# B&R Automation Studio project TD52 (part 70)

```iecst
END_TYPE
TYPE
END_TYPE
```

#### lib_properties.txt
```
For manual assignment to hardware configuration please
add the following additional include directories:

\Logical\MATLAB_includes\R2021b\

And the following additional build options:

-lm -D MODEL=Gen2_ref -D NUMST=1 -D NCSTATES=0 -D HAVESTDIO -D MODEL_HAS_DYNAMICALLY_LOADED_SFCNS=0 -D CLASSIC_INTERFACE=0 -D ALLOCATIONFCN=0 -D TID01EQ=0 -D TERMFCN=1 -D ONESTEPFCN=1 -D MAT_FILE=0 -D MULTI_INSTANCE_CODE=1 -D INTEGER_CODE=0 -D MT=0
```

#### rtGetInf.c
```c
/********************************************************************
 * COPYRIGHT -- B&R Industrial Automation GmbH
 ********************************************************************
 * Program: Gen2_ref
 * File: rtGetInf.c
 * Author: 105055527
 * Last modified by: kelleto00
 * Created: Wed Apr 16 13:02:53 2008
 * Last modified: Wed Oct 09 10:01:33 2024
 * Model Version: 4.14.00.04
 * Description: V4.10.00.01, 01-09-2020 Keller, Ke Estimator, additive LS factor, Ptraj SpeedCtrl, LVRT Freeze HLCi
   V4.10.00.01, 02-10-2020 Keller, bugfix HLCi p2srefLX init, BDC_lib: change Inf to 1e7
   V4.10.00.01, 13-11-2020 Keller, bugfix LXcorr T2s/ZZP, LSLff damping, dbgOut for Leanox WG compensation
   V4.10.00.01, 27-01-2021 Keller, Lx WGV compensation: no reset in island mode, addition before skipfire compensation
   V4.10.00.01, 02-02-2021 Keller, initialization lambda estimation with rLam_Start
   V4.11.00.01, 28-05-2021 Keller, Gas Quality Change (GQC) Improvements, LHV estimator output
   V4.11.00.01, 05-11-2021 Keller, Bugfix BDC: worksplit offset, optionally Nset instead of Nnom, rN_Eng_LRskipF
   V4.12.00.01, 10-02-2021 Keller, SpeedCtrl2.0 TU Wien: Disturbance Estimator, LQR incl. droop & leanox
   V4.12.00.02, 23-05-2022 Arnold, Leanox point C in low load
   V4.12.00.02, 09-06-2022 Kafka, add external skip fire input for isolated and grid parallel operation
   V4.12.00.03, 15-09-2022 Keller, add power trajectory to HLCi for extended LQR (Droop setpoint)
   V4.12.00.04, 12-10-2022 Keller, add gas flow comp. factor for rejections
   V4.12.00.05, 13-10-2022 Keller, power filter for static skipfire in island mode
   V4.12.00.06, 15-11-2022 Keller, Ke adaptation with disturbance observer
   V4.13.00.01, 15-11-2022 Keller, FDC: R_mix output, HLCi: R_mix for Ke
   V4.13.00.02, 10-07-2023 Keller, interpolation of LHV, rho_gas and Lmin
   V4.13.00.03, 10-07-2023 Keller, load dependent gas dosage delay
   V4.13.00.04, 11-09-2023 Keller, D-part FSM, bugfix dPTV ramp
   V4.13.00.05, 27-02-2024 Keller, Filter outputs without bSS
   V4.13.00.06, 10-04-2024 Keller, bugfix leanox manual mode with bSepEmisCtrl
   V4.14.00.01, 01-07-2024 Keller, iNskip_LRfor Ke calculation
   V4.14.00.02, 17-09-2024 Keller, Use actual speed for observer disturbance dg (Gen2_ref/HLC_Island (HLC_Island_ref)/iLQR_SF/Ref LQR)
   V4.14.00.03, 30-09-2024 Keller, LR gas flow compensation possible without actuator saturation
   V4.14.00.04, 02-10-2024 Keller, Limit derivative power setpoint for FSM
 * modified Comment:
 ********************************************************************
 * Implementation of program Gen2_ref
 ********************************************************************
 * Generated with B&R Automation Studio Target for Simulink V6.7.1
 * (ERT based)
 ********************************************************************/

/*
 * Abstract:
 *      Function to initialize non-finite, Inf
 */
#include "rtGetInf.h"

/*  Defines */
#define NumBitsPerChar                 8U

/*  Data Types */

/**************************** GLOBAL DATA *************************************/
/*  Definitions */

/*  Declarations  */

/***************************** FILE SCOPE DATA ********************************/

/*************************** FUNCTIONS ****************************************/

/*
 * Initialize rtInf needed by the generated code.
 * Inf is initialized as non-signaling. Assumes IEEE.
 */
real_T rtGetInf(void)
{
  size_t bitsPerReal = sizeof(real_T) * (NumBitsPerChar);
  real_T inf = 0.0;
  if (bitsPerReal == 32U) {
    inf = rtGetInfF();
  } else {
    union {
      LittleEndianIEEEDouble bitVal;
      real_T fltVal;
    } tmpVal;

    tmpVal.bitVal.words.wordH = 0x7FF00000U;
    tmpVal.bitVal.words.wordL = 0x00000000U;
    inf = tmpVal.fltVal;
  }

  return inf;
}

/*
 * Initialize rtInfF needed by the generated code.
 * Inf is initialized as non-signaling. Assumes IEEE.
 */
real32_T rtGetInfF(void)
{
  IEEESingle infF;
  infF.wordL.wordLuint = 0x7F800000U;
  return infF.wordL.wordLreal;
}

/*
 * Initialize rtMinusInf needed by the generated code.
 * Inf is initialized as non-signaling. Assumes IEEE.
 */
real_T rtGetMinusInf(void)
{
  size_t bitsPerReal = sizeof(real_T) * (NumBitsPerChar);
  real_T minf = 0.0;
  if (bitsPerReal == 32U) {
    minf = rtGetMinusInfF();
  } else {
    union {
      LittleEndianIEEEDouble bitVal;
      real_T fltVal;
    } tmpVal;

    tmpVal.bitVal.words.wordH = 0xFFF00000U;
    tmpVal.bitVal.words.wordL = 0x00000000U;
    minf = tmpVal.fltVal;
  }

  return minf;
}

/*
 * Initialize rtMinusInfF needed by the generated code.
 * Inf is initialized as non-signaling. Assumes IEEE.
 */
real32_T rtGetMinusInfF(void)
{
  IEEESingle minfF;
  minfF.wordL.wordLuint = 0xFF800000U;
  return minfF.wordL.wordLreal;
}

/*======================== TOOL VERSION INFORMATION ==========================*
 * MATLAB 9.11 (R2021b)14-May-2021                                            *
 * Simulink 10.4 (R2021b)14-May-2021                                          *
 * Simulink Coder 9.6 (R2021b)14-May-2021                                     *
 * Embedded Coder 7.7 (R2021b)14-May-2021                                     *
 * Stateflow 10.5 (R2021b)14-May-2021                                         *
 *============================================================================*/

/*======================= LICENSE IN USE INFORMATION =========================*
 * control_toolbox                                                            *
 * matlab                                                                     *
 * matlab_coder                                                               *
 * real-time_workshop                                                         *
 * rtw_embedded_coder                                                         *
 * simulink                                                                   *
 *============================================================================*/
```

#### rtGetInf.h
```c
/********************************************************************
 * COPYRIGHT -- B&R Industrial Automation GmbH
 ********************************************************************
 * Program: Gen2_ref
 * File: rtGetInf.h
 * Author: 105055527
 * Last modified by: kelleto00
 * Created: Wed Apr 16 13:02:53 2008
 * Last modified: Wed Oct 09 10:01:33 2024
 * Model Version: 4.14.00.04
 * Description: V4.10.00.01, 01-09-2020 Keller, Ke Estimator, additive LS factor, Ptraj SpeedCtrl, LVRT Freeze HLCi
   V4.10.00.01, 02-10-2020 Keller, bugfix HLCi p2srefLX init, BDC_lib: change Inf to 1e7
   V4.10.00.01, 13-11-2020 Keller, bugfix LXcorr T2s/ZZP, LSLff damping, dbgOut for Leanox WG compensation
   V4.10.00.01, 27-01-2021 Keller, Lx WGV compensation: no reset in island mode, addition before skipfire compensation
   V4.10.00.01, 02-02-2021 Keller, initialization lambda estimation with rLam_Start
   V4.11.00.01, 28-05-2021 Keller, Gas Quality Change (GQC) Improvements, LHV estimator output
   V4.11.00.01, 05-11-2021 Keller, Bugfix BDC: worksplit offset, optionally Nset instead of Nnom, rN_Eng_LRskipF
   V4.12.00.01, 10-02-2021 Keller, SpeedCtrl2.0 TU Wien: Disturbance Estimator, LQR incl. droop & leanox
   V4.12.00.02, 23-05-2022 Arnold, Leanox point C in low load
   V4.12.00.02, 09-06-2022 Kafka, add external skip fire input for isolated and grid parallel operation
   V4.12.00.03, 15-09-2022 Keller, add power trajectory to HLCi for extended LQR (Droop setpoint)
   V4.12.00.04, 12-10-2022 Keller, add gas flow comp. factor for rejections
   V4.12.00.05, 13-10-2022 Keller, power filter for static skipfire in island mode
   V4.12.00.06, 15-11-2022 Keller, Ke adaptation with disturbance observer
   V4.13.00.01, 15-11-2022 Keller, FDC: R_mix output, HLCi: R_mix for Ke
   V4.13.00.02, 10-07-2023 Keller, interpolation of LHV, rho_gas and Lmin
   V4.13.00.03, 10-07-2023 Keller, load dependent gas dosage delay
   V4.13.00.04, 11-09-2023 Keller, D-part FSM, bugfix dPTV ramp
   V4.13.00.05, 27-02-2024 Keller, Filter outputs without bSS
   V4.13.00.06, 10-04-2024 Keller, bugfix leanox manual mode with bSepEmisCtrl
   V4.14.00.01, 01-07-2024 Keller, iNskip_LRfor Ke calculation
   V4.14.00.02, 17-09-2024 Keller, Use actual speed for observer disturbance dg (Gen2_ref/HLC_Island (HLC_Island_ref)/iLQR_SF/Ref LQR)
   V4.14.00.03, 30-09-2024 Keller, LR gas flow compensation possible without actuator saturation
   V4.14.00.04, 02-10-2024 Keller, Limit derivative power setpoint for FSM
 * modified Comment:
 ********************************************************************
 * Header for program Gen2_ref
 ********************************************************************
 * Generated with B&R Automation Studio Target for Simulink V6.7.1
 * (ERT based)
 ********************************************************************/

#ifndef RTW_HEADER_rtGetInf_h_
#define RTW_HEADER_rtGetInf_h_
#include <stddef.h>
#include "rtwtypes.h"
#include "rt_nonfinite.h"
#ifndef MIN
#define MIN(a,b)                       ((a) < (b) ? (a) : (b))
#endif

#ifndef MAX
#define MAX(a,b)                       ((a) > (b) ? (a) : (b))
#endif

#ifndef AST_ROUND
#define AST_ROUND(x)                   ((x)>=0?(long long)((x)+0.5):(long long)((x)-0.5))
#endif

extern real_T rtGetInf(void);
extern real32_T rtGetInfF(void);
extern real_T rtGetMinusInf(void);
extern real32_T rtGetMinusInfF(void);

#endif                                 /* RTW_HEADER_rtGetInf_h_ */
```

#### rtGetNaN.c
```c
/********************************************************************
 * COPYRIGHT -- B&R Industrial Automation GmbH
 ********************************************************************
 * Program: Gen2_ref
 * File: rtGetNaN.c
 * Author: 105055527
 * Last modified by: kelleto00
 * Created: Wed Apr 16 13:02:53 2008
 * Last modified: Wed Oct 09 10:01:33 2024
 * Model Version: 4.14.00.04
 * Description: V4.10.00.01, 01-09-2020 Keller, Ke Estimator, additive LS factor, Ptraj SpeedCtrl, LVRT Freeze HLCi
   V4.10.00.01, 02-10-2020 Keller, bugfix HLCi p2srefLX init, BDC_lib: change Inf to 1e7
   V4.10.00.01, 13-11-2020 Keller, bugfix LXcorr T2s/ZZP, LSLff damping, dbgOut for Leanox WG compensation
   V4.10.00.01, 27-01-2021 Keller, Lx WGV compensation: no reset in island mode, addition before skipfire compensation
   V4.10.00.01, 02-02-2021 Keller, initialization lambda estimation with rLam_Start
   V4.11.00.01, 28-05-2021 Keller, Gas Quality Change (GQC) Improvements, LHV estimator output
   V4.11.00.01, 05-11-2021 Keller, Bugfix BDC: worksplit offset, optionally Nset instead of Nnom, rN_Eng_LRskipF
   V4.12.00.01, 10-02-2021 Keller, SpeedCtrl2.0 TU Wien: Disturbance Estimator, LQR incl. droop & leanox
   V4.12.00.02, 23-05-2022 Arnold, Leanox point C in low load
   V4.12.00.02, 09-06-2022 Kafka, add external skip fire input for isolated and grid parallel operation
   V4.12.00.03, 15-09-2022 Keller, add power trajectory to HLCi for extended LQR (Droop setpoint)
   V4.12.00.04, 12-10-2022 Keller, add gas flow comp. factor for rejections
   V4.12.00.05, 13-10-2022 Keller, power filter for static skipfire in island mode
   V4.12.00.06, 15-11-2022 Keller, Ke adaptation with disturbance observer
   V4.13.00.01, 15-11-2022 Keller, FDC: R_mix output, HLCi: R_mix for Ke
   V4.13.00.02, 10-07-2023 Keller, interpolation of LHV, rho_gas and Lmin
   V4.13.00.03, 10-07-2023 Keller, load dependent gas dosage delay
   V4.13.00.04, 11-09-2023 Keller, D-part FSM, bugfix dPTV ramp
   V4.13.00.05, 27-02-2024 Keller, Filter outputs without bSS
   V4.13.00.06, 10-04-2024 Keller, bugfix leanox manual mode with bSepEmisCtrl
   V4.14.00.01, 01-07-2024 Keller, iNskip_LRfor Ke calculation
   V4.14.00.02, 17-09-2024 Keller, Use actual speed for observer disturbance dg (Gen2_ref/HLC_Island (HLC_Island_ref)/iLQR_SF/Ref LQR)
   V4.14.00.03, 30-09-2024 Keller, LR gas flow compensation possible without actuator saturation
   V4.14.00.04, 02-10-2024 Keller, Limit derivative power setpoint for FSM
 * modified Comment:
 ********************************************************************
 * Implementation of program Gen2_ref
 ********************************************************************
 * Generated with B&R Automation Studio Target for Simulink V6.7.1
 * (ERT based)
 ********************************************************************/

/*
 * Abstract:
 *      Function to initialize non-finite, NaN
 */
#include "rtGetNaN.h"

/*  Defines */
#define NumBitsPerChar                 8U

/*  Data Types */

/**************************** GLOBAL DATA *************************************/
/*  Definitions */

/*  Declarations  */

/***************************** FILE SCOPE DATA ********************************/

/*************************** FUNCTIONS ****************************************/

/*
 * Initialize rtNaN needed by the generated code.
 * NaN is initialized as non-signaling. Assumes IEEE.
 */
real_T rtGetNaN(void)
{
  size_t bitsPerReal = sizeof(real_T) * (NumBitsPerChar);
  real_T nan = 0.0;
  if (bitsPerReal == 32U) {
    nan = rtGetNaNF();
  } else {
    union {
      LittleEndianIEEEDouble bitVal;
      real_T fltVal;
    } tmpVal;

    tmpVal.bitVal.words.wordH = 0xFFF80000U;
    tmpVal.bitVal.words.wordL = 0x00000000U;
    nan = tmpVal.fltVal;
  }

  return nan;
}

/*
 * Initialize rtNaNF needed by the generated code.
 * NaN is initialized as non-signaling. Assumes IEEE.
 */
real32_T rtGetNaNF(void)
{
  IEEESingle nanF = { { 0.0F } };

  nanF.wordL.wordLuint = 0xFFC00000U;
  return nanF.wordL.wordLreal;
}

/*======================== TOOL VERSION INFORMATION ==========================*
 * MATLAB 9.11 (R2021b)14-May-2021                                            *
 * Simulink 10.4 (R2021b)14-May-2021                                          *
 * Simulink Coder 9.6 (R2021b)14-May-2021                                     *
 * Embedded Coder 7.7 (R2021b)14-May-2021                                     *
 * Stateflow 10.5 (R2021b)14-May-2021                                         *
 *============================================================================*/

/*======================= LICENSE IN USE INFORMATION =========================*
 * control_toolbox                                                            *
 * matlab                                                                     *
 * matlab_coder                                                               *
 * real-time_workshop                                                         *
 * rtw_embedded_coder                                                         *
 * simulink                                                                   *
 *============================================================================*/
```

#### rtGetNaN.h
```c
/********************************************************************
 * COPYRIGHT -- B&R Industrial Automation GmbH
 ********************************************************************
 * Program: Gen2_ref
 * File: rtGetNaN.h
 * Author: 105055527
 * Last modified by: kelleto00
 * Created: Wed Apr 16 13:02:53 2008
 * Last modified: Wed Oct 09 10:01:33 2024
 * Model Version: 4.14.00.04
 * Description: V4.10.00.01, 01-09-2020 Keller, Ke Estimator, additive LS factor, Ptraj SpeedCtrl, LVRT Freeze HLCi
   V4.10.00.01, 02-10-2020 Keller, bugfix HLCi p2srefLX init, BDC_lib: change Inf to 1e7
   V4.10.00.01, 13-11-2020 Keller, bugfix LXcorr T2s/ZZP, LSLff damping, dbgOut for Leanox WG compensation
   V4.10.00.01, 27-01-2021 Keller, Lx WGV compensation: no reset in island mode, addition before skipfire compensation
   V4.10.00.01, 02-02-2021 Keller, initialization lambda estimation with rLam_Start
   V4.11.00.01, 28-05-2021 Keller, Gas Quality Change (GQC) Improvements, LHV estimator output
   V4.11.00.01, 05-11-2021 Keller, Bugfix BDC: worksplit offset, optionally Nset instead of Nnom, rN_Eng_LRskipF
   V4.12.00.01, 10-02-2021 Keller, SpeedCtrl2.0 TU Wien: Disturbance Estimator, LQR incl. droop & leanox
   V4.12.00.02, 23-05-2022 Arnold, Leanox point C in low load
   V4.12.00.02, 09-06-2022 Kafka, add external skip fire input for isolated and grid parallel operation
   V4.12.00.03, 15-09-2022 Keller, add power trajectory to HLCi for extended LQR (Droop setpoint)
   V4.12.00.04, 12-10-2022 Keller, add gas flow comp. factor for rejections
   V4.12.00.05, 13-10-2022 Keller, power filter for static skipfire in island mode
   V4.12.00.06, 15-11-2022 Keller, Ke adaptation with disturbance observer
   V4.13.00.01, 15-11-2022 Keller, FDC: R_mix output, HLCi: R_mix for Ke
   V4.13.00.02, 10-07-2023 Keller, interpolation of LHV, rho_gas and Lmin
   V4.13.00.03, 10-07-2023 Keller, load dependent gas dosage delay
   V4.13.00.04, 11-09-2023 Keller, D-part FSM, bugfix dPTV ramp
   V4.13.00.05, 27-02-2024 Keller, Filter outputs without bSS
   V4.13.00.06, 10-04-2024 Keller, bugfix leanox manual mode with bSepEmisCtrl
   V4.14.00.01, 01-07-2024 Keller, iNskip_LRfor Ke calculation
   V4.14.00.02, 17-09-2024 Keller, Use actual speed for observer disturbance dg (Gen2_ref/HLC_Island (HLC_Island_ref)/iLQR_SF/Ref LQR)
   V4.14.00.03, 30-09-2024 Keller, LR gas flow compensation possible without actuator saturation
   V4.14.00.04, 02-10-2024 Keller, Limit derivative power setpoint for FSM
 * modified Comment:
 ********************************************************************
 * Header for program Gen2_ref
 ********************************************************************
 * Generated with B&R Automation Studio Target for Simulink V6.7.1
 * (ERT based)
 ********************************************************************/

#ifndef RTW_HEADER_rtGetNaN_h_
#define RTW_HEADER_rtGetNaN_h_
#include <stddef.h>
#include "rtwtypes.h"
#include "rt_nonfinite.h"
#ifndef MIN
#define MIN(a,b)                       ((a) < (b) ? (a) : (b))
#endif

#ifndef MAX
#define MAX(a,b)                       ((a) > (b) ? (a) : (b))
#endif

#ifndef AST_ROUND
#define AST_ROUND(x)                   ((x)>=0?(long long)((x)+0.5):(long long)((x)-0.5))
#endif

extern real_T rtGetNaN(void);
extern real32_T rtGetNaNF(void);

#endif                                 /* RTW_HEADER_rtGetNaN_h_ */
```

#### rt_defines.h
```c
/********************************************************************
 * COPYRIGHT -- B&R Industrial Automation GmbH
 ********************************************************************
 * Program: Gen2_ref
 * File: rt_defines.h
 * Author: 105055527
 * Last modified by: kelleto00
 * Created: Wed Apr 16 13:02:53 2008
 * Last modified: Wed Oct 09 10:01:33 2024
 * Model Version: 4.14.00.04
 * Description: V4.10.00.01, 01-09-2020 Keller, Ke Estimator, additive LS factor, Ptraj SpeedCtrl, LVRT Freeze HLCi
   V4.10.00.01, 02-10-2020 Keller, bugfix HLCi p2srefLX init, BDC_lib: change Inf to 1e7
   V4.10.00.01, 13-11-2020 Keller, bugfix LXcorr T2s/ZZP, LSLff damping, dbgOut for Leanox WG compensation
   V4.10.00.01, 27-01-2021 Keller, Lx WGV compensation: no reset in island mode, addition before skipfire compensation
   V4.10.00.01, 02-02-2021 Keller, initialization lambda estimation with rLam_Start
   V4.11.00.01, 28-05-2021 Keller, Gas Quality Change (GQC) Improvements, LHV estimator output
   V4.11.00.01, 05-11-2021 Keller, Bugfix BDC: worksplit offset, optionally Nset instead of Nnom, rN_Eng_LRskipF
   V4.12.00.01, 10-02-2021 Keller, SpeedCtrl2.0 TU Wien: Disturbance Estimator, LQR incl. droop & leanox
   V4.12.00.02, 23-05-2022 Arnold, Leanox point C in low load
   V4.12.00.02, 09-06-2022 Kafka, add external skip fire input for isolated and grid parallel operation
   V4.12.00.03, 15-09-2022 Keller, add power trajectory to HLCi for extended LQR (Droop setpoint)
   V4.12.00.04, 12-10-2022 Keller, add gas flow comp. factor for rejections
   V4.12.00.05, 13-10-2022 Keller, power filter for static skipfire in island mode
   V4.12.00.06, 15-11-2022 Keller, Ke adaptation with disturbance observer
   V4.13.00.01, 15-11-2022 Keller, FDC: R_mix output, HLCi: R_mix for Ke
   V4.13.00.02, 10-07-2023 Keller, interpolation of LHV, rho_gas and Lmin
   V4.13.00.03, 10-07-2023 Keller, load dependent gas dosage delay
   V4.13.00.04, 11-09-2023 Keller, D-part FSM, bugfix dPTV ramp
   V4.13.00.05, 27-02-2024 Keller, Filter outputs without bSS
   V4.13.00.06, 10-04-2024 Keller, bugfix leanox manual mode with bSepEmisCtrl
   V4.14.00.01, 01-07-2024 Keller, iNskip_LRfor Ke calculation
   V4.14.00.02, 17-09-2024 Keller, Use actual speed for observer disturbance dg (Gen2_ref/HLC_Island (HLC_Island_ref)/iLQR_SF/Ref LQR)
   V4.14.00.03, 30-09-2024 Keller, LR gas flow compensation possible without actuator saturation
   V4.14.00.04, 02-10-2024 Keller, Limit derivative power setpoint for FSM
 * modified Comment:
 ********************************************************************
 * Header for program Gen2_ref
 ********************************************************************
 * Generated with B&R Automation Studio Target for Simulink V6.7.1
 * (ERT based)
 ********************************************************************/

#ifndef RTW_HEADER_rt_defines_h_
#define RTW_HEADER_rt_defines_h_
#ifndef MIN
#define MIN(a,b)                       ((a) < (b) ? (a) : (b))
#endif

#ifndef MAX
#define MAX(a,b)                       ((a) > (b) ? (a) : (b))
#endif

#ifndef AST_ROUND
#define AST_ROUND(x)                   ((x)>=0?(long long)((x)+0.5):(long long)((x)-0.5))
#endif

/*===========*
 * Constants *
 *===========*/
#define RT_PI                          3.14159265358979323846
#define RT_PIF                         3.1415927F
#define RT_LN_10                       2.30258509299404568402
#define RT_LN_10F                      2.3025851F
#define RT_LOG10E                      0.43429448190325182765
#define RT_LOG10EF                     0.43429449F
#define RT_E                           2.7182818284590452354
#define RT_EF                          2.7182817F

/*
 * UNUSED_PARAMETER(x)
 *   Used to specify that a function parameter (argument) is required but not
 *   accessed by the function body.
 */
#ifndef UNUSED_PARAMETER
#if defined(__LCC__)
#define UNUSED_PARAMETER(x)                                      /* do nothing */
#else

/*
 * This is the semi-ANSI standard way of indicating that an
 * unused function parameter is required.
 */
#define UNUSED_PARAMETER(x)            (void) (x)
#endif
#endif
#endif                                 /* RTW_HEADER_rt_defines_h_ */
```

#### rt_nonfinite.c
```c
/********************************************************************
 * COPYRIGHT -- B&R Industrial Automation GmbH
 ********************************************************************
 * Program: Gen2_ref
 * File: rt_nonfinite.c
 * Author: 105055527
 * Last modified by: kelleto00
 * Created: Wed Apr 16 13:02:53 2008
 * Last modified: Wed Oct 09 10:01:33 2024
 * Model Version: 4.14.00.04
 * Description: V4.10.00.01, 01-09-2020 Keller, Ke Estimator, additive LS factor, Ptraj SpeedCtrl, LVRT Freeze HLCi
   V4.10.00.01, 02-10-2020 Keller, bugfix HLCi p2srefLX init, BDC_lib: change Inf to 1e7
   V4.10.00.01, 13-11-2020 Keller, bugfix LXcorr T2s/ZZP, LSLff damping, dbgOut for Leanox WG compensation
   V4.10.00.01, 27-01-2021 Keller, Lx WGV compensation: no reset in island mode, addition before skipfire compensation
   V4.10.00.01, 02-02-2021 Keller, initialization lambda estimation with rLam_Start
   V4.11.00.01, 28-05-2021 Keller, Gas Quality Change (GQC) Improvements, LHV estimator output
   V4.11.00.01, 05-11-2021 Keller, Bugfix BDC: worksplit offset, optionally Nset instead of Nnom, rN_Eng_LRskipF
   V4.12.00.01, 10-02-2021 Keller, SpeedCtrl2.0 TU Wien: Disturbance Estimator, LQR incl. droop & leanox
   V4.12.00.02, 23-05-2022 Arnold, Leanox point C in low load
   V4.12.00.02, 09-06-2022 Kafka, add external skip fire input for isolated and grid parallel operation
   V4.12.00.03, 15-09-2022 Keller, add power trajectory to HLCi for extended LQR (Droop setpoint)
   V4.12.00.04, 12-10-2022 Keller, add gas flow comp. factor for rejections
   V4.12.00.05, 13-10-2022 Keller, power filter for static skipfire in island mode
   V4.12.00.06, 15-11-2022 Keller, Ke adaptation with disturbance observer
   V4.13.00.01, 15-11-2022 Keller, FDC: R_mix output, HLCi: R_mix for Ke
   V4.13.00.02, 10-07-2023 Keller, interpolation of LHV, rho_gas and Lmin
   V4.13.00.03, 10-07-2023 Keller, load dependent gas dosage delay
   V4.13.00.04, 11-09-2023 Keller, D-part FSM, bugfix dPTV ramp
   V4.13.00.05, 27-02-2024 Keller, Filter outputs without bSS
   V4.13.00.06, 10-04-2024 Keller, bugfix leanox manual mode with bSepEmisCtrl
   V4.14.00.01, 01-07-2024 Keller, iNskip_LRfor Ke calculation
   V4.14.00.02, 17-09-2024 Keller, Use actual speed for observer disturbance dg (Gen2_ref/HLC_Island (HLC_Island_ref)/iLQR_SF/Ref LQR)
   V4.14.00.03, 30-09-2024 Keller, LR gas flow compensation possible without actuator saturation
   V4.14.00.04, 02-10-2024 Keller, Limit derivative power setpoint for FSM
 * modified Comment:
 ********************************************************************
 * Implementation of program Gen2_ref
 ********************************************************************
 * Generated with B&R Automation Studio Target for Simulink V6.7.1
 * (ERT based)
 ********************************************************************/

/*
 * Abstract:
 *      Function to initialize non-finites,
 *      (Inf, NaN and -Inf).
 */
#include "rt_nonfinite.h"
#include "rtGetNaN.h"
#include "rtGetInf.h"

/*  Defines */
#define NumBitsPerChar                 8U

/*  Data Types */

/**************************** GLOBAL DATA *************************************/
/*  Definitions */

/*  Declarations  */
real_T rtInf;
real_T rtMinusInf;
real_T rtNaN;
real32_T rtInfF;
real32_T rtMinusInfF;
real32_T rtNaNF;

/***************************** FILE SCOPE DATA ********************************/

/*************************** FUNCTIONS ****************************************/

/*
 * Initialize the rtInf, rtMinusInf, and rtNaN needed by the
 * generated code. NaN is initialized as non-signaling. Assumes IEEE.
 */
void rt_InitInfAndNaN(size_t realSize)
{
  (void) (realSize);
  rtNaN = rtGetNaN();
  rtNaNF = rtGetNaNF();
  rtInf = rtGetInf();
  rtInfF = rtGetInfF();
  rtMinusInf = rtGetMinusInf();
  rtMinusInfF = rtGetMinusInfF();
}

/* Test if value is infinite */
boolean_T rtIsInf(real_T value)
{
  return (boolean_T)((value==rtInf || value==rtMinusInf) ? 1U : 0U);
}

/* Test if single-precision value is infinite */
boolean_T rtIsInfF(real32_T value)
{
  return (boolean_T)(((value)==rtInfF || (value)==rtMinusInfF) ? 1U : 0U);
}

/* Test if value is not a number */
boolean_T rtIsNaN(real_T value)
{
  boolean_T result = (boolean_T) 0;
  size_t bitsPerReal = sizeof(real_T) * (NumBitsPerChar);
  if (bitsPerReal == 32U) {
    result = rtIsNaNF((real32_T)value);
  } else {
    union {
      LittleEndianIEEEDouble bitVal;
      real_T fltVal;
    } tmpVal;

    tmpVal.fltVal = value;
    result = (boolean_T)((tmpVal.bitVal.words.wordH & 0x7FF00000) == 0x7FF00000 &&
                         ( (tmpVal.bitVal.words.wordH & 0x000FFFFF) != 0 ||
                          (tmpVal.bitVal.words.wordL != 0) ));
  }

  return result;
}

/* Test if single-precision value is not a number */
boolean_T rtIsNaNF(real32_T value)
{
  IEEESingle tmp;
  tmp.wordL.wordLreal = value;
  return (boolean_T)( (tmp.wordL.wordLuint & 0x7F800000) == 0x7F800000 &&
                     (tmp.wordL.wordLuint & 0x007FFFFF) != 0 );
}

/*======================== TOOL VERSION INFORMATION ==========================*
 * MATLAB 9.11 (R2021b)14-May-2021                                            *
 * Simulink 10.4 (R2021b)14-May-2021                                          *
 * Simulink Coder 9.6 (R2021b)14-May-2021                                     *
 * Embedded Coder 7.7 (R2021b)14-May-2021                                     *
 * Stateflow 10.5 (R2021b)14-May-2021                                         *
 *============================================================================*/

/*======================= LICENSE IN USE INFORMATION =========================*
 * control_toolbox                                                            *
 * matlab                                                                     *
 * matlab_coder                                                               *
 * real-time_workshop                                                         *
 * rtw_embedded_coder                                                         *
 * simulink                                                                   *
 *============================================================================*/
```

#### rt_nonfinite.h
```c
/********************************************************************
 * COPYRIGHT -- B&R Industrial Automation GmbH
 ********************************************************************
 * Program: Gen2_ref
 * File: rt_nonfinite.h
 * Author: 105055527
 * Last modified by: kelleto00
 * Created: Wed Apr 16 13:02:53 2008
 * Last modified: Wed Oct 09 10:01:33 2024
 * Model Version: 4.14.00.04
 * Description: V4.10.00.01, 01-09-2020 Keller, Ke Estimator, additive LS factor, Ptraj SpeedCtrl, LVRT Freeze HLCi
   V4.10.00.01, 02-10-2020 Keller, bugfix HLCi p2srefLX init, BDC_lib: change Inf to 1e7
   V4.10.00.01, 13-11-2020 Keller, bugfix LXcorr T2s/ZZP, LSLff damping, dbgOut for Leanox WG compensation
   V4.10.00.01, 27-01-2021 Keller, Lx WGV compensation: no reset in island mode, addition before skipfire compensation
   V4.10.00.01, 02-02-2021 Keller, initialization lambda estimation with rLam_Start
   V4.11.00.01, 28-05-2021 Keller, Gas Quality Change (GQC) Improvements, LHV estimator output
   V4.11.00.01, 05-11-2021 Keller, Bugfix BDC: worksplit offset, optionally Nset instead of Nnom, rN_Eng_LRskipF
   V4.12.00.01, 10-02-2021 Keller, SpeedCtrl2.0 TU Wien: Disturbance Estimator, LQR incl. droop & leanox
   V4.12.00.02, 23-05-2022 Arnold, Leanox point C in low load
   V4.12.00.02, 09-06-2022 Kafka, add external skip fire input for isolated and grid parallel operation
   V4.12.00.03, 15-09-2022 Keller, add power trajectory to HLCi for extended LQR (Droop setpoint)
   V4.12.00.04, 12-10-2022 Keller, add gas flow comp. factor for rejections
   V4.12.00.05, 13-10-2022 Keller, power filter for static skipfire in island mode
   V4.12.00.06, 15-11-2022 Keller, Ke adaptation with disturbance observer
   V4.13.00.01, 15-11-2022 Keller, FDC: R_mix output, HLCi: R_mix for Ke
   V4.13.00.02, 10-07-2023 Keller, interpolation of LHV, rho_gas and Lmin
   V4.13.00.03, 10-07-2023 Keller, load dependent gas dosage delay
   V4.13.00.04, 11-09-2023 Keller, D-part FSM, bugfix dPTV ramp
   V4.13.00.05, 27-02-2024 Keller, Filter outputs without bSS
   V4.13.00.06, 10-04-2024 Keller, bugfix leanox manual mode with bSepEmisCtrl
   V4.14.00.01, 01-07-2024 Keller, iNskip_LRfor Ke calculation
   V4.14.00.02, 17-09-2024 Keller, Use actual speed for observer disturbance dg (Gen2_ref/HLC_Island (HLC_Island_ref)/iLQR_SF/Ref LQR)
   V4.14.00.03, 30-09-2024 Keller, LR gas flow compensation possible without actuator saturation
   V4.14.00.04, 02-10-2024 Keller, Limit derivative power setpoint for FSM
 * modified Comment:
 ********************************************************************
 * Header for program Gen2_ref
 ********************************************************************
 * Generated with B&R Automation Studio Target for Simulink V6.7.1
 * (ERT based)
 ********************************************************************/

#ifndef RTW_HEADER_rt_nonfinite_h_
#define RTW_HEADER_rt_nonfinite_h_
#include <stddef.h>
#include "rtwtypes.h"
#ifndef MIN
#define MIN(a,b)                       ((a) < (b) ? (a) : (b))
#endif

#ifndef MAX
#define MAX(a,b)                       ((a) > (b) ? (a) : (b))
#endif

#ifndef AST_ROUND
#define AST_ROUND(x)                   ((x)>=0?(long long)((x)+0.5):(long long)((x)-0.5))
#endif

extern real_T rtInf;
extern real_T rtMinusInf;
extern real_T rtNaN;
extern real32_T rtInfF;
extern real32_T rtMinusInfF;
extern real32_T rtNaNF;
extern void rt_InitInfAndNaN(size_t realSize);
extern boolean_T rtIsInf(real_T value);
extern boolean_T rtIsInfF(real32_T value);
extern boolean_T rtIsNaN(real_T value);
extern boolean_T rtIsNaNF(real32_T value);
typedef struct {
  struct {
    uint32_T wordH;
    uint32_T wordL;
  } words;
} BigEndianIEEEDouble;

typedef struct {
  struct {
    uint32_T wordL;
    uint32_T wordH;
  } words;
} LittleEndianIEEEDouble;

typedef struct {
  union {
    real32_T wordLreal;
    uint32_T wordLuint;
  } wordL;
} IEEESingle;

#endif                                 /* RTW_HEADER_rt_nonfinite_h_ */
```

#### rtwtypes.h
```c
/********************************************************************
 * COPYRIGHT -- B&R Industrial Automation GmbH
 ********************************************************************
 * Program: Gen2_ref
 * File: rtwtypes.h
 * Author: 105055527
 * Last modified by: kelleto00
 * Created: Wed Apr 16 13:02:53 2008
 * Last modified: Wed Oct 09 10:01:33 2024
 * Model Version: 4.14.00.04
 * Description: V4.10.00.01, 01-09-2020 Keller, Ke Estimator, additive LS factor, Ptraj SpeedCtrl, LVRT Freeze HLCi
   V4.10.00.01, 02-10-2020 Keller, bugfix HLCi p2srefLX init, BDC_lib: change Inf to 1e7
   V4.10.00.01, 13-11-2020 Keller, bugfix LXcorr T2s/ZZP, LSLff damping, dbgOut for Leanox WG compensation
   V4.10.00.01, 27-01-2021 Keller, Lx WGV compensation: no reset in island mode, addition before skipfire compensation
   V4.10.00.01, 02-02-2021 Keller, initialization lambda estimation with rLam_Start
   V4.11.00.01, 28-05-2021 Keller, Gas Quality Change (GQC) Improvements, LHV estimator output
   V4.11.00.01, 05-11-2021 Keller, Bugfix BDC: worksplit offset, optionally Nset instead of Nnom, rN_Eng_LRskipF
   V4.12.00.01, 10-02-2021 Keller, SpeedCtrl2.0 TU Wien: Disturbance Estimator, LQR incl. droop & leanox
   V4.12.00.02, 23-05-2022 Arnold, Leanox point C in low load
   V4.12.00.02, 09-06-2022 Kafka, add external skip fire input for isolated and grid parallel operation
   V4.12.00.03, 15-09-2022 Keller, add power trajectory to HLCi for extended LQR (Droop setpoint)
   V4.12.00.04, 12-10-2022 Keller, add gas flow comp. factor for rejections
   V4.12.00.05, 13-10-2022 Keller, power filter for static skipfire in island mode
   V4.12.00.06, 15-11-2022 Keller, Ke adaptation with disturbance observer
   V4.13.00.01, 15-11-2022 Keller, FDC: R_mix output, HLCi: R_mix for Ke
   V4.13.00.02, 10-07-2023 Keller, interpolation of LHV, rho_gas and Lmin
   V4.13.00.03, 10-07-2023 Keller, load dependent gas dosage delay
   V4.13.00.04, 11-09-2023 Keller, D-part FSM, bugfix dPTV ramp
   V4.13.00.05, 27-02-2024 Keller, Filter outputs without bSS
   V4.13.00.06, 10-04-2024 Keller, bugfix leanox manual mode with bSepEmisCtrl
   V4.14.00.01, 01-07-2024 Keller, iNskip_LRfor Ke calculation
   V4.14.00.02, 17-09-2024 Keller, Use actual speed for observer disturbance dg (Gen2_ref/HLC_Island (HLC_Island_ref)/iLQR_SF/Ref LQR)
   V4.14.00.03, 30-09-2024 Keller, LR gas flow compensation possible without actuator saturation
   V4.14.00.04, 02-10-2024 Keller, Limit derivative power setpoint for FSM
 * modified Comment:
 ********************************************************************
 * Header for program Gen2_ref
 ********************************************************************
 * Generated with B&R Automation Studio Target for Simulink V6.7.1
 * (ERT based)
 ********************************************************************/

#ifndef RTWTYPES_H
#define RTWTYPES_H

/* Logical type definitions */
#if (!defined(__cplusplus))
#ifndef false
#define false                          (0U)
#endif

#ifndef true
#define true                           (1U)
#endif
#endif

/*=======================================================================*
 * Target hardware information
 *   Device type: Intel->x86/Pentium
 *   Number of bits:     char:   8    short:   16    long:  32
 *                       long:  32
 *                       native word size:  32
 *   Byte ordering: LittleEndian
 *   Signed integer division rounds to: Zero
 *   Shift right on a signed integer as arithmetic shift: on
 *=======================================================================*/

/*=======================================================================*
 * Fixed width word size data types:                                     *
 *   int8_T, int16_T, int32_T     - signed 8, 16, or 32 bit integers     *
 *   uint8_T, uint16_T, uint32_T  - unsigned 8, 16, or 32 bit integers   *
 *   real32_T, real64_T           - 32 and 64 bit floating point numbers *
 *=======================================================================*/
typedef signed char int8_T;
typedef unsigned char uint8_T;
typedef short int16_T;
typedef unsigned short uint16_T;
typedef long int32_T;
typedef unsigned long uint32_T;
typedef float real32_T;
typedef double real64_T;

/*===========================================================================*
 * Generic type definitions: boolean_T, char_T, byte_T, int_T, uint_T,       *
 *                           real_T, time_T, ulong_T.                        *
 *===========================================================================*/
typedef double real_T;
typedef double time_T;
typedef unsigned char boolean_T;
typedef long int_T;
typedef unsigned long uint_T;
typedef unsigned long ulong_T;
typedef char char_T;
typedef unsigned char uchar_T;
typedef char_T byte_T;

/*=======================================================================*
 * Min and Max:                                                          *
 *   int8_T, int16_T, int32_T     - signed 8, 16, or 32 bit integers     *
 *   uint8_T, uint16_T, uint32_T  - unsigned 8, 16, or 32 bit integers   *
 *=======================================================================*/
#define MAX_int8_T                     ((int8_T)(127))
#define MIN_int8_T                     ((int8_T)(-128))
#define MAX_uint8_T                    ((uint8_T)(255U))
#define MAX_int16_T                    ((int16_T)(32767))
#define MIN_int16_T                    ((int16_T)(-32768))
#define MAX_uint16_T                   ((uint16_T)(65535U))
#define MAX_int32_T                    ((int32_T)(2147483647))
#define MIN_int32_T                    ((int32_T)(-2147483647-1))
#define MAX_uint32_T                   ((uint32_T)(0xFFFFFFFFU))

/* Block D-Work pointer type */
typedef void * pointer_T;

#endif                                 /* RTWTYPES_H */

#ifndef MIN
#define MIN(a,b)                       ((a) < (b) ? (a) : (b))
#endif

#ifndef MAX
#define MAX(a,b)                       ((a) > (b) ? (a) : (b))
#endif

#ifndef AST_ROUND
#define AST_ROUND(x)                   ((x)>=0?(long long)((x)+0.5):(long long)((x)-0.5))
#endif
```

#### zero_crossing_types.h
```c
/********************************************************************
 * COPYRIGHT -- B&R Industrial Automation GmbH
 ********************************************************************
 * Program: Gen2_ref
 * File: zero_crossing_types.h
 * Author: 105055527
 * Last modified by: kelleto00
 * Created: Wed Apr 16 13:02:53 2008
 * Last modified: Wed Oct 09 10:01:33 2024
 * Model Version: 4.14.00.04
 * Description: V4.10.00.01, 01-09-2020 Keller, Ke Estimator, additive LS factor, Ptraj SpeedCtrl, LVRT Freeze HLCi
   V4.10.00.01, 02-10-2020 Keller, bugfix HLCi p2srefLX init, BDC_lib: change Inf to 1e7
   V4.10.00.01, 13-11-2020 Keller, bugfix LXcorr T2s/ZZP, LSLff damping, dbgOut for Leanox WG compensation
   V4.10.00.01, 27-01-2021 Keller, Lx WGV compensation: no reset in island mode, addition before skipfire compensation
   V4.10.00.01, 02-02-2021 Keller, initialization lambda estimation with rLam_Start
   V4.11.00.01, 28-05-2021 Keller, Gas Quality Change (GQC) Improvements, LHV estimator output
   V4.11.00.01, 05-11-2021 Keller, Bugfix BDC: worksplit offset, optionally Nset instead of Nnom, rN_Eng_LRskipF
   V4.12.00.01, 10-02-2021 Keller, SpeedCtrl2.0 TU Wien: Disturbance Estimator, LQR incl. droop & leanox
   V4.12.00.02, 23-05-2022 Arnold, Leanox point C in low load
   V4.12.00.02, 09-06-2022 Kafka, add external skip fire input for isolated and grid parallel operation
   V4.12.00.03, 15-09-2022 Keller, add power trajectory to HLCi for extended LQR (Droop setpoint)
   V4.12.00.04, 12-10-2022 Keller, add gas flow comp. factor for rejections
   V4.12.00.05, 13-10-2022 Keller, power filter for static skipfire in island mode
   V4.12.00.06, 15-11-2022 Keller, Ke adaptation with disturbance observer
   V4.13.00.01, 15-11-2022 Keller, FDC: R_mix output, HLCi: R_mix for Ke
   V4.13.00.02, 10-07-2023 Keller, interpolation of LHV, rho_gas and Lmin
   V4.13.00.03, 10-07-2023 Keller, load dependent gas dosage delay
   V4.13.00.04, 11-09-2023 Keller, D-part FSM, bugfix dPTV ramp
   V4.13.00.05, 27-02-2024 Keller, Filter outputs without bSS
   V4.13.00.06, 10-04-2024 Keller, bugfix leanox manual mode with bSepEmisCtrl
   V4.14.00.01, 01-07-2024 Keller, iNskip_LRfor Ke calculation
   V4.14.00.02, 17-09-2024 Keller, Use actual speed for observer disturbance dg (Gen2_ref/HLC_Island (HLC_Island_ref)/iLQR_SF/Ref LQR)
   V4.14.00.03, 30-09-2024 Keller, LR gas flow compensation possible without actuator saturation
   V4.14.00.04, 02-10-2024 Keller, Limit derivative power setpoint for FSM
 * modified Comment:
 ********************************************************************
 * Header for program Gen2_ref
 ********************************************************************
 * Generated with B&R Automation Studio Target for Simulink V6.7.1
 * (ERT based)
 ********************************************************************/

#ifndef ZERO_CROSSING_TYPES_H
#define ZERO_CROSSING_TYPES_H
#include "rtwtypes.h"

/* Trigger directions: falling, either, and rising */
typedef enum {
  FALLING_ZERO_CROSSING = -1,
  ANY_ZERO_CROSSING = 0,
  RISING_ZERO_CROSSING = 1
} ZCDirection;

/* Previous state of a trigger signal */
typedef uint8_T ZCSigState;

/* Initial value of a trigger zero crossing signal */
#define UNINITIALIZED_ZCSIG            0x03U
#define NEG_ZCSIG                      0x02U
#define POS_ZCSIG                      0x01U
#define ZERO_ZCSIG                     0x00U

/* Current state of a trigger signal */
typedef enum {
  FALLING_ZCEVENT = -1,
  NO_ZCEVENT = 0,
  RISING_ZCEVENT = 1
} ZCEventType;

#endif                                 /* ZERO_CROSSING_TYPES_H */

#ifndef MIN
#define MIN(a,b)                       ((a) < (b) ? (a) : (b))
#endif

#ifndef MAX
#define MAX(a,b)                       ((a) > (b) ? (a) : (b))
#endif

#ifndef AST_ROUND
#define AST_ROUND(x)                   ((x)>=0?(long long)((x)+0.5):(long long)((x)-0.5))
#endif
```

### Library Logical/EngineController/Lib_EC/lPFPDR (ANSIC)

#### lPFPDR.fun
```iecst
FUNCTION_BLOCK PFPDR
  VAR_INPUT
    ssMethodType: SINT;
  END_VAR  VAR_INPUT
        in : tPFPDR_In; (**)
  END_VAR
  VAR_INPUT
        par : tPFPDR_Para; (**)
  END_VAR
 VAR_OUTPUT
        out : tPFPDR_Out; (**)
  END_VAR
 VAR_OUTPUT
        dbg : tPFPDR_Dbg; (**)
  END_VAR
	VAR
		bur_BlockIO_AC_PFPDR : BlockIO_AC_PFPDR;
	END_VAR
	VAR
		bur_D_Work_AC_PFPDR : D_Work_AC_PFPDR;
	END_VAR
END_FUNCTION_BLOCK
```

#### lPFPDR.typ
```iecst
TYPE

   tPFPDR_Dbg : STRUCT
        rT_Sampling : REAL; (*Cycle Time, for which PFPDR was compiled*)
        rCA_IP_aDR : ARRAY[0..24] OF REAL; (*Ignition profile snapshot after duration run [°CA]*)
        rCA_IP_bDR : ARRAY[0..24] OF REAL; (*Ignition profile snapshot before duration run [°CA]*)
        rCA_IP_aDR_Avg : REAL; (*average of ignition profile snapshot after duration run [°CA]*)
        rCA_IP_bDR_Avg : REAL; (*average of ignition profile snapshot before duration run [°CA]*)
        bAbort_DR : ARRAY[0..2] OF BOOL; (*PFPDR Abort conditions*)
    END_STRUCT;

   tPFPDR_In : STRUCT
        bStartTrigger : BOOL; (*TRUE = starts PFPDR routine if in steady state*)
        rT_EG_Act : ARRAY[0..24] OF REAL; (*Actual exhaust gas temperature [°C]*)
        rCA_IP_Act : ARRAY[0..24] OF REAL; (*Actual ignition point [°CA]*)
        rCA_IP_Set : REAL; (*Ignition setpoint [°CA]*)
        rCA_Knck_Red : ARRAY[0..24] OF REAL; (*Ignition point reduction due knocking [°CA]*)
        iNum_Cyl : USINT; (*Number of cylinders*)
        rT_EG_Avg : REAL; (*Actual average exhaust gas temperature [°C]*)
        bMisfLim : BOOL; (*Misfire Limit reached, goto lambda decrease steps*)
        bManAbort : BOOL; (*Manual Abort PFPDR and EGTSR*)
        bReset : BOOL; (*Resets the Integrators in the Steady State machine*)
        rLam_Act : REAL; (*Actual Lambda of Engine [Lambda]*)
        bPFPDR_Profile : BOOL; (*is the engine currently running a PFPDR Profile? if Yes the engine is old*)
        rPos_CBV : REAL; (*position of compressor by pass [-]*)
        bSteadyState : BOOL; (*TRUE = starts PFPDR routine if in start trigger*)
    END_STRUCT;

   tPFPDR_Out : STRUCT
        iState : ARRAY[0..1] OF INT; (*Statemachine states [0]: 0=IDLE, 1=PFPDR, 2=EGT; [1]: 0= no Substate, 1=Start, 2=Ignition, 3=Lambda, 4=Save, 5=LamReturn, 6= IgnReturn*)
        rLam_DR_Offs : REAL; (*Lambda offset during detection run [Lambda]*)
        rCA_IP_DR_Offs : REAL; (*Ignition point offset during detection run [°CA]*)
        bLeanox_Man : BOOL; (*Leanox has to be taken in manual mode if TRUE*)
        rCA_IP_DR_Profile : ARRAY[0..24] OF REAL; (*Calculated ignition point offset from detection run [°CA]*)
        rCA_IP_EGT_Profile : ARRAY[0..24] OF REAL; (*Calculated ignition point offset from EGT deviation [°CA]*)
        bPFPDR_act : BOOL; (*PFPDR is active*)
        bEGTSR_act : BOOL; (*EGTSR is active*)
        bZYLOPT_OFF : BOOL; (*force ZYLOPT OFF if true*)
    END_STRUCT;

   tPFPDR_Para : STRUCT
        rCA_IP_MaxLim : REAL; (*Ignition point maximum limit eg. type4 = 27 [°CA]*)
        rT_EG_DevLim : REAL; (*Exhaust gas temperature deviation limit from average, e.g. 10 [°C]*)
        rCA_IP_EGT : REAL; (*Ignition point offset if exhaust gas deviation occurs eg. 1 [°CA]*)
        rTi_EGT_Delay : REAL; (*Time delay before EGT devation routine starts eg. 180 [s]*)
        rLam_DR_Lim : REAL; (*maximum delta lamba during duration run [lambda]*)
        rLam_DR_SR : REAL; (*lambda slew rate during duration run [lambda/s]*)
        rLam_DR_SR_Return : REAL; (*lambda slew rate after duration run [lambda/s]*)
        rCA_IP_DR_SR : REAL; (*ignition point slew rate during duration run [°CA/s]*)
        rCA_IP_DR_SR_Return : REAL; (*ignition point slew rate after duration run [°CA/s]*)
        rPos_CBV_Opt : REAL; (*optimized position of compressor by pass [-]*)
        rPos_CBV_Hys : REAL; (*hysterese position of compressor by pass [-]*)
        rT_Abort_Delay : REAL; (*delay of abort [s]*)
        rT_Abort_Filter : REAL; (*filter of abort [s]*)
    END_STRUCT;
END_TYPE
TYPE
rtB_TON_AC_PFPDR : STRUCT
	LogicalOperator3 : BOOL;
END_STRUCT;
rtDW_TON_AC_PFPDR : STRUCT
	DiscreteTimeIntegrator_DSTATE : REAL;
	DiscreteTimeIntegrator_PrevRese : SINT;
END_STRUCT;
BlockIO_AC_PFPDR : STRUCT
	BusInput1 : tPFPDR_In;
	BusConversion_InsertedFor_BusOu : tPFPDR_Out;
	BusConversion_InsertedFor_Bus_c : tPFPDR_Dbg;
	BusInput : tPFPDR_Para;
	rT_EG_Act : ARRAY[0..24] OF REAL;
	rCA_IP_Act : ARRAY[0..24] OF REAL;
	rLam_Act : REAL;
	rCA_IP_MaxLim : REAL;
	rT_EG_DevLim : REAL;
	rCA_IP_EGT : REAL;
	Divide : REAL;
	Product : REAL;
	Product1 : REAL;
	Product2 : REAL;
	Product3 : REAL;
	rCA_IP_aDR : ARRAY[0..24] OF REAL;
	rCA_IP_bDR_Avg : REAL;
	rCA_IP_DR_Offs : REAL;
	rLam_DR_Offs : REAL;
	rCA_IP_bDR : ARRAY[0..24] OF REAL;
	rCA_IP_aDR_Max : REAL;
	rCA_IP_EGT_Offs : ARRAY[0..24] OF REAL;
	rCA_IP_aDR_Offs : ARRAY[0..24] OF REAL;
	iState : INT;
	iSubState : INT;
	u4Cylinder : USINT;
	bStartTrigger : BOOL;
	bMisfLim : BOOL;
	bManAbort : BOOL;
	bReset : BOOL;
	bSteadyState : BOOL;
	UnitDelay : BOOL;
	UnitDelay1 : BOOL;
	UnitDelay2 : BOOL;
	bLeanox_Man : BOOL;
	bPFPDR_active : BOOL;
	bEGTSR_active : BOOL;
	TON1 : rtB_TON_AC_PFPDR;
	TON : rtB_TON_AC_PFPDR;
END_STRUCT;
D_Work_AC_PFPDR : STRUCT
	iCnt : REAL;
	rLam_bDR : REAL;
	rCA_IgnP_Act_Filt : ARRAY[0..24] OF REAL;
	rCnt_Filt : REAL;
	UnitDelay_DSTATE : BOOL;
	UnitDelay1_DSTATE : BOOL;
	UnitDelay2_DSTATE : BOOL;
	UnitDelay2_DSTATE_l : BOOL;
	is_active_c6_AC_PFPDR : USINT;
	is_c6_AC_PFPDR : USINT;
	is_DetectionRun : USINT;
	bDR_Done : BOOL;
	bDR_Lam : BOOL;
	bEGT_Done : BOOL;
	TON1 : rtDW_TON_AC_PFPDR;
	TON : rtDW_TON_AC_PFPDR;
END_STRUCT;
END_TYPE
```

#### AC_PFPDR.h
```c
/********************************************************************
 * COPYRIGHT -- Bernecker + Rainer Industrie-Elektronik Ges.m.b.H.
 ********************************************************************
 * Program: AC_PFPDR
 * File: AC_PFPDR.h
 * Author: 502423184
 * Created: Fri Apr 24 12:55:11 2015
 ********************************************************************
 * Header for program AC_PFPDR
 ********************************************************************
 * Generated with B&R Automation Studio Target for Simulink V4.2
 * (ERT based)
 ********************************************************************/

#ifndef RTW_HEADER_AC_PFPDR_h_
#define RTW_HEADER_AC_PFPDR_h_
#ifndef AC_PFPDR_COMMON_INCLUDES_
# define AC_PFPDR_COMMON_INCLUDES_
#include <math.h>
#include "rtwtypes.h"
#endif                                 /* AC_PFPDR_COMMON_INCLUDES_ */

#include "AC_PFPDR_types.h"
#include "lPFPDR.h"

/* Macros for accessing real-time model data structure */
#ifndef rtmGetErrorStatus
# define rtmGetErrorStatus(rtm)        ((void*) 0)
#endif

#ifndef rtmSetErrorStatus
# define rtmSetErrorStatus(rtm, val)   ((void) 0)
#endif

#ifndef rtmGetStopRequested
# define rtmGetStopRequested(rtm)      ((void*) 0)
#endif

#ifndef MIN
#define MIN(a,b)                       ((a) < (b) ? (a) : (b))
#endif

#ifndef MAX
#define MAX(a,b)                       ((a) > (b) ? (a) : (b))
#endif

/* Block signals for system '<S9>/TON' */

/* Block states (auto storage) for system '<S9>/TON' */

/* Block signals (auto storage) */

/* Block states (auto storage) for system '<Root>' */

/* Model entry point functions */
extern void AC_PFPDR_initialize(struct PFPDR* inst);
extern void AC_PFPDR_step(BlockIO_AC_PFPDR *AC_PFPDR_B, D_Work_AC_PFPDR
  *AC_PFPDR_DWork, struct PFPDR* inst);
extern void AC_PFPDR_terminate(struct PFPDR* inst);

/*-
 * The generated code includes comments that allow you to trace directly
 * back to the appropriate location in the model.  The basic format
 * is <system>/block_name, where system is the system number (uniquely
 * assigned by Simulink) and block_name is the name of the block.
 *
 * Use the MATLAB hilite_system command to trace the generated code back
 * to the model.  For example,
 *
 * hilite_system('<S3>')    - opens system 3
 * hilite_system('<S3>/Kp') - opens and selects block Kp which resides in S3
 *
 * Here is the system hierarchy for this model
 *
 * '<Root>' : 'AC_PFPDR'
 * '<S1>'   : 'AC_PFPDR/SimuBlock'
 * '<S2>'   : 'AC_PFPDR/SimuBlock/PFPDR_Autocode'
 * '<S3>'   : 'AC_PFPDR/SimuBlock/PFPDR_Autocode/Environment Controller'
 * '<S4>'   : 'AC_PFPDR/SimuBlock/PFPDR_Autocode/Environment Controller1'
 * '<S5>'   : 'AC_PFPDR/SimuBlock/PFPDR_Autocode/PFPDR'
 * '<S6>'   : 'AC_PFPDR/SimuBlock/PFPDR_Autocode/PFPDR/Abort Conditions'
 * '<S7>'   : 'AC_PFPDR/SimuBlock/PFPDR_Autocode/PFPDR/Chart (MATLAB)'
 * '<S8>'   : 'AC_PFPDR/SimuBlock/PFPDR_Autocode/PFPDR/Hysterese'
 * '<S9>'   : 'AC_PFPDR/SimuBlock/PFPDR_Autocode/PFPDR/Time Delay'
 * '<S10>'  : 'AC_PFPDR/SimuBlock/PFPDR_Autocode/PFPDR/Abort Conditions/Abort Condition 1'
 * '<S11>'  : 'AC_PFPDR/SimuBlock/PFPDR_Autocode/PFPDR/Abort Conditions/Abort Condition 2'
 * '<S12>'  : 'AC_PFPDR/SimuBlock/PFPDR_Autocode/PFPDR/Abort Conditions/Abort Condition 3'
 * '<S13>'  : 'AC_PFPDR/SimuBlock/PFPDR_Autocode/PFPDR/Time Delay/TON'
 * '<S14>'  : 'AC_PFPDR/SimuBlock/PFPDR_Autocode/PFPDR/Time Delay/TON1'
 * '<S15>'  : 'AC_PFPDR/SimuBlock/PFPDR_Autocode/PFPDR/Time Delay/TON/Data Type Conversion Inherited'
 * '<S16>'  : 'AC_PFPDR/SimuBlock/PFPDR_Autocode/PFPDR/Time Delay/TON1/Data Type Conversion Inherited'
 */
#endif                                 /* RTW_HEADER_AC_PFPDR_h_ */
```

#### AC_PFPDR_private.h
```c
/********************************************************************
 * COPYRIGHT -- Bernecker + Rainer Industrie-Elektronik Ges.m.b.H.
 ********************************************************************
 * Program: AC_PFPDR
 * File: AC_PFPDR_private.h
 * Author: 502423184
 * Created: Fri Apr 24 12:55:11 2015
 ********************************************************************
 * Header for program AC_PFPDR
 ********************************************************************
 * Generated with B&R Automation Studio Target for Simulink V4.2
 * (ERT based)
 ********************************************************************/

#ifndef RTW_HEADER_AC_PFPDR_private_h_
#define RTW_HEADER_AC_PFPDR_private_h_
#include "rtwtypes.h"
#include <bur/plctypes.h>
#ifndef __RTWTYPES_H__
#error This file requires rtwtypes.h to be included
#else
#ifdef TMWTYPES_PREVIOUSLY_INCLUDED
#error This file requires rtwtypes.h to be included before tmwtypes.h
#else

/* Check for inclusion of an incorrect version of rtwtypes.h */
#ifndef RTWTYPES_ID_C08S16I32L32N32F1
#error This code was generated with a different "rtwtypes.h" than the file included
#endif                                 /* RTWTYPES_ID_C08S16I32L32N32F1 */
#endif                                 /* TMWTYPES_PREVIOUSLY_INCLUDED */
#endif                                 /* __RTWTYPES_H__ */

#ifndef MIN
#define MIN(a,b)                       ((a) < (b) ? (a) : (b))
#endif

#ifndef MAX
#define MAX(a,b)                       ((a) > (b) ? (a) : (b))
#endif

extern real_T rt_roundd(real_T u, struct PFPDR* inst);

/* Exported functions */
extern void AC_PFPDR_TON(boolean_T rtu_IN, real32_T rtu_PT, rtB_TON_AC_PFPDR
  *localB, rtDW_TON_AC_PFPDR *localDW, struct PFPDR* inst);

#endif                                 /* RTW_HEADER_AC_PFPDR_private_h_ */
```

#### AC_PFPDR_types.h
```c
/********************************************************************
 * COPYRIGHT -- Bernecker + Rainer Industrie-Elektronik Ges.m.b.H.
 ********************************************************************
 * Program: AC_PFPDR
 * File: AC_PFPDR_types.h
 * Author: 502423184
 * Created: Fri Apr 24 12:55:11 2015
 ********************************************************************
 * Header for program AC_PFPDR
 ********************************************************************
 * Generated with B&R Automation Studio Target for Simulink V4.2
 * (ERT based)
 ********************************************************************/

#ifndef RTW_HEADER_AC_PFPDR_types_h_
#define RTW_HEADER_AC_PFPDR_types_h_
#include "rtwtypes.h"
#ifndef MIN
#define MIN(a,b)                       ((a) < (b) ? (a) : (b))
#endif

#ifndef MAX
#define MAX(a,b)                       ((a) > (b) ? (a) : (b))
#endif

#endif                                 /* RTW_HEADER_AC_PFPDR_types_h_ */
```

#### rtwtypes.h
```c
/********************************************************************
 * COPYRIGHT -- Bernecker + Rainer Industrie-Elektronik Ges.m.b.H.
 ********************************************************************
 * Program: AC_PFPDR
 * File: rtwtypes.h
 * Author: 502423184
 * Created: Fri Apr 24 12:55:11 2015
 ********************************************************************
 * Header for program AC_PFPDR
 ********************************************************************
 * Generated with B&R Automation Studio Target for Simulink V4.2
 * (ERT based)
 ********************************************************************/

#ifndef __RTWTYPES_H__
#define __RTWTYPES_H__
#ifndef TRUE
# define TRUE                          (1U)
#endif

#ifndef FALSE
# define FALSE                         (0U)
#endif

#ifndef __TMWTYPES__
#define __TMWTYPES__
#include <limits.h>

/*=======================================================================*
 * Target hardware information
 *   Device type: Intel->x86/Pentium
 *   Number of bits:     char:   8    short:   16    long:  32
 *                       long:  32
 *                       native word size:  32
 *   Byte ordering: LittleEndian
 *   Signed integer division rounds to: Zero
 *   Shift right on a signed integer as arithmetic shift: on
 *=======================================================================*/

/*=======================================================================*
 * Fixed width word size data types:                                     *
 *   int8_T, int16_T, int32_T     - signed 8, 16, or 32 bit integers     *
 *   uint8_T, uint16_T, uint32_T  - unsigned 8, 16, or 32 bit integers   *
 *   real32_T, real64_T           - 32 and 64 bit floating point numbers *
 *=======================================================================*/
typedef signed char int8_T;
typedef unsigned char uint8_T;
typedef short int16_T;
typedef unsigned short uint16_T;
typedef long int32_T;
typedef unsigned long uint32_T;
typedef float real32_T;
typedef double real64_T;

/*===========================================================================*
 * Generic type definitions: real_T, time_T, boolean_T, int_T, uint_T,       *
 *                           ulong_T, char_T and byte_T.                     *
 *===========================================================================*/
typedef double real_T;
typedef double time_T;
typedef unsigned char boolean_T;
typedef long int_T;
typedef unsigned long uint_T;
typedef unsigned long ulong_T;
typedef char char_T;
typedef unsigned char uchar_T;
typedef char_T byte_T;

/*=======================================================================*
 * Min and Max:                                                          *
 *   int8_T, int16_T, int32_T     - signed 8, 16, or 32 bit integers     *
 *   uint8_T, uint16_T, uint32_T  - unsigned 8, 16, or 32 bit integers   *
 *=======================================================================*/
#define MAX_int8_T                     ((int8_T)(127))
#define MIN_int8_T                     ((int8_T)(-128))
#define MAX_uint8_T                    ((uint8_T)(255U))
#define MIN_uint8_T                    ((uint8_T)(0U))
#define MAX_int16_T                    ((int16_T)(32767))
#define MIN_int16_T                    ((int16_T)(-32768))
#define MAX_uint16_T                   ((uint16_T)(65535U))
#define MIN_uint16_T                   ((uint16_T)(0U))
#define MAX_int32_T                    ((int32_T)(2147483647))
#define MIN_int32_T                    ((int32_T)(-2147483647-1))
#define MAX_uint32_T                   ((uint32_T)(0xFFFFFFFFU))
#define MIN_uint32_T                   ((uint32_T)(0U))

/* Logical type definitions */
#if (!defined(__cplusplus)) && (!defined(__true_false_are_keywords))
#  ifndef false
#   define false                       (0U)
#  endif

#  ifndef true
#   define true                        (1U)
#  endif
#endif

/*
 * Simulink Coder assumes the code is compiled on a target using a 2's complement representation
 * for signed integer values.
 */
#if ((SCHAR_MIN + 1) != -SCHAR_MAX)
#error "This code must be compiled using a 2's complement representation for signed integer values"
#endif

/* This ID is used to detect inclusion of an incompatible rtwtypes.h */
#define RTWTYPES_ID_C08S16I32L32N32F1
#else                                  /* __TMWTYPES__ */
#define TMWTYPES_PREVIOUSLY_INCLUDED
#endif                                 /* __TMWTYPES__ */

/* Block D-Work pointer type */
typedef void * pointer_T;

/* Simulink specific types */
#ifndef __SIMSTRUC_TYPES_H__
#define __SIMSTRUC_TYPES_H__

/* Trigger directions: falling, either, and rising */
typedef enum {
  FALLING_ZERO_CROSSING = -1,
  ANY_ZERO_CROSSING = 0,
  RISING_ZERO_CROSSING = 1
} ZCDirection;

/* Previous state of a trigger signal */
typedef uint8_T ZCSigState;

/* Initial value of a trigger zero crossing signal */
#define UNINITIALIZED_ZCSIG            0x03U
#define NEG_ZCSIG                      0x02U
#define POS_ZCSIG                      0x01U
#define ZERO_ZCSIG                     0x00U

/* Current state of a trigger signal */
typedef enum {
  FALLING_ZCEVENT = -1,
  NO_ZCEVENT = 0,
  RISING_ZCEVENT = 1
} ZCEventType;

#endif                                 /* __SIMSTRUC_TYPES_H__ */
#endif                                 /* __RTWTYPES_H__ */

#ifndef MIN
#define MIN(a,b)                       ((a) < (b) ? (a) : (b))
#endif

#ifndef MAX
#define MAX(a,b)                       ((a) > (b) ? (a) : (b))
#endif
```

#### AC_PFPDR.c
```c
/********************************************************************
 * COPYRIGHT -- Bernecker + Rainer Industrie-Elektronik Ges.m.b.H.
 ********************************************************************
 * Program: AC_PFPDR
 * File: AC_PFPDR.c
 * Author: 502423184
 * Created: Fri Apr 24 12:55:11 2015
 ********************************************************************
 * Implementation of program AC_PFPDR
 ********************************************************************
 * Generated with B&R Automation Studio Target for Simulink V4.2
 * (ERT based)
 ********************************************************************/
#include "AC_PFPDR.h"
#include "AC_PFPDR_private.h"

/*  Defines */

/* Named constants for Chart: '<S5>/Chart (MATLAB)' */
#define AC_PFPDR_IN_Abort              ((uint8_T)1U)
#define AC_PFPDR_IN_Detection          ((uint8_T)1U)
#define AC_PFPDR_IN_DetectionRun       ((uint8_T)2U)
#define AC_PFPDR_IN_EGTSR              ((uint8_T)3U)
#define AC_PFPDR_IN_IDLE               ((uint8_T)4U)
#define AC_PFPDR_IN_IgnitionPoint      ((uint8_T)2U)
#define AC_PFPDR_IN_IgnpointReturn     ((uint8_T)3U)
#define AC_PFPDR_IN_Lambda             ((uint8_T)4U)
#define AC_PFPDR_IN_LambdaReturn       ((uint8_T)5U)
#define AC_PFPDR_IN_NO_ACTIVE_CHILD    ((uint8_T)0U)
#define AC_PFPDR_IN_SaveProfile        ((uint8_T)6U)

/*  Data Types */

/**************************** GLOBAL DATA *************************************/
/*  Definitions */

/*  Declarations  */

/* Forward declaration for local functions */
static void AC_PFP_enter_atomic_SaveProfile(struct BlockIO_AC_PFPDR *AC_PFPDR_B,
  struct D_Work_AC_PFPDR *AC_PFPDR_DWork, struct PFPDR* inst);
static void AC_PFPDR_exit_atomic_EGTSR(struct BlockIO_AC_PFPDR *AC_PFPDR_B, struct PFPDR* inst);

/***************************** FILE SCOPE DATA ********************************/

/*************************** FUNCTIONS ****************************************/

/*
 * Output and update for atomic system:
 *    '<S9>/TON'
 *    '<S9>/TON1'
 */
void AC_PFPDR_TON(boolean_T rtu_IN, real32_T rtu_PT, rtB_TON_AC_PFPDR *localB,
                  rtDW_TON_AC_PFPDR *localDW, struct PFPDR* inst)
{
  /* local block i/o variables */
  boolean_T rtb_LogicalOperator2;
  boolean_T rtb_RelationalOperator;

  /* Logic: '<S13>/Logical Operator2' */
  rtb_LogicalOperator2 = !rtu_IN;

  /* DiscreteIntegrator: '<S13>/Discrete-Time Integrator' */
  if (rtb_LogicalOperator2 || (localDW->DiscreteTimeIntegrator_PrevRese != 0)) {
    localDW->DiscreteTimeIntegrator_DSTATE = 0.0F;
  }

  /* RelationalOperator: '<S13>/Relational Operator' incorporates:
   *  DiscreteIntegrator: '<S13>/Discrete-Time Integrator'
   */
  rtb_RelationalOperator = (localDW->DiscreteTimeIntegrator_DSTATE >= rtu_PT);

  /* Logic: '<S13>/Logical Operator3' */
  localB->LogicalOperator3 = (rtb_RelationalOperator && rtu_IN);

  /* Update for DiscreteIntegrator: '<S13>/Discrete-Time Integrator' incorporates:
   *  DataTypeConversion: '<S15>/Conversion'
   *  Logic: '<S13>/Logical Operator'
   *  Logic: '<S13>/Logical Operator1'
   */
  if (!rtb_LogicalOperator2) {
    localDW->DiscreteTimeIntegrator_DSTATE += (real32_T)
      ((!rtb_RelationalOperator) && rtu_IN) * 0.01F;
  }

  if (rtb_LogicalOperator2) {
    localDW->DiscreteTimeIntegrator_PrevRese = 1;
  } else {
    localDW->DiscreteTimeIntegrator_PrevRese = 0;
  }

  /* End of Update for DiscreteIntegrator: '<S13>/Discrete-Time Integrator' */
}

/* Function for Chart: '<S5>/Chart (MATLAB)' */
static void AC_PFP_enter_atomic_SaveProfile(struct BlockIO_AC_PFPDR *AC_PFPDR_B,
  struct D_Work_AC_PFPDR *AC_PFPDR_DWork, struct PFPDR* inst)
{
  uint8_T iCyl;
  int32_T i;

  /* Entry 'SaveProfile': '<S7>:74' */
  AC_PFPDR_B->iSubState = 4;
  for (i = 0; i < 25; i++) {
    AC_PFPDR_B->rCA_IP_aDR[i] = AC_PFPDR_DWork->rCA_IgnP_Act_Filt[i] /
      AC_PFPDR_DWork->rCnt_Filt;
  }

  /* Store actual Ignition Points */
  AC_PFPDR_B->rCA_IP_aDR_Max = 0.0F;
  i = (int32_T)((uint32_T)AC_PFPDR_B->u4Cylinder + 1U);
  if ((uint32_T)i > 255U) {
    i = 255;
  }

  for (iCyl = 2U; iCyl <= (uint8_T)i; iCyl = (uint8_T)((uint32_T)iCyl + 1U)) {
    if (AC_PFPDR_B->rCA_IP_aDR_Max < AC_PFPDR_B->rCA_IP_aDR[iCyl - 1]) {
      AC_PFPDR_B->rCA_IP_aDR_Max = AC_PFPDR_B->rCA_IP_aDR[iCyl - 1];
    }
  }

  i = (int32_T)((uint32_T)AC_PFPDR_B->u4Cylinder + 1U);
  if ((uint32_T)i > 255U) {
    i = 255;
  }

  for (iCyl = 2U; iCyl <= (uint8_T)i; iCyl = (uint8_T)((uint32_T)iCyl + 1U)) {
    AC_PFPDR_B->rCA_IP_aDR_Offs[iCyl - 1] = AC_PFPDR_B->rCA_IP_aDR[iCyl - 1] +
      -AC_PFPDR_B->rCA_IP_aDR_Max;
  }
}

/* Function for Chart: '<S5>/Chart (MATLAB)' */
static void AC_PFPDR_exit_atomic_EGTSR(struct BlockIO_AC_PFPDR *AC_PFPDR_B, struct PFPDR* inst)
{
  uint8_T iCyl;
  real32_T rT_EG_Avg;
  int32_T i;
  real32_T rT_EG_Avg_0;

  /* Exit 'EGTSR': '<S7>:5' */
  /* rT_EG_Avg = sum(rT_EG_Act(2:iNum_Cyl+1))/iNum_Cyl; */
  rT_EG_Avg = 0.0F;
  i = (int32_T)((uint32_T)AC_PFPDR_B->u4Cylinder + 1U);
  if ((uint32_T)i > 255U) {
    i = 255;
  }

  for (iCyl = 2U; iCyl <= (uint8_T)i; iCyl = (uint8_T)((uint32_T)iCyl + 1U)) {
    rT_EG_Avg += AC_PFPDR_B->rT_EG_Act[iCyl - 1];
  }

  rT_EG_Avg /= (real32_T)AC_PFPDR_B->u4Cylinder;

  /* too cold cylinders: */
  /* too hot cylinders: */
  rT_EG_Avg_0 = rT_EG_Avg + AC_PFPDR_B->rT_EG_DevLim;
  for (i = 0; i < 25; i++) {
    AC_PFPDR_B->rCA_IP_EGT_Offs[i] = (real32_T)((AC_PFPDR_B->rT_EG_Act[i] <
      rT_EG_Avg - AC_PFPDR_B->rT_EG_DevLim) && (AC_PFPDR_B->rT_EG_Act[i] >
      rT_EG_Avg - 50.0F)) * -AC_PFPDR_B->rCA_IP_EGT;
    AC_PFPDR_B->rCA_IP_EGT_Offs[i] += (real32_T)((AC_PFPDR_B->rT_EG_Act[i] >
      rT_EG_Avg_0) && (AC_PFPDR_B->rT_EG_Act[i] < rT_EG_Avg + 50.0F)) *
      AC_PFPDR_B->rCA_IP_EGT;
  }
}

real_T rt_roundd(real_T u, struct PFPDR* inst)
{
  real_T y;
  if (fabs(u) < 4.503599627370496E+15) {
    if (u >= 0.5) {
      y = floor(u + 0.5);
    } else if (u > -0.5) {
      y = 0.0;
    } else {
      y = ceil(u - 0.5);
    }
  } else {
    y = u;
  }

  return y;
}

/* Model step function */
void AC_PFPDR_step(struct BlockIO_AC_PFPDR *AC_PFPDR_B, struct D_Work_AC_PFPDR *AC_PFPDR_DWork, struct PFPDR* inst)
{
  /* local block i/o variables */
  real32_T rtb_rT_Abort_Delay;
  real32_T rtb_Subtract;
  boolean_T rtb_Abort;
  real32_T rCA_IP_Max;
  uint8_T rtb_iNum_Cyl;
  boolean_T rtb_abort1;
  boolean_T rtb_abort2;
  boolean_T rtb_abort3;
  int32_T rtb_Switch;
  int32_T i;

  /* S-Function (bur_bus_in): '<S2>/Bus Input1' */
  AC_PFPDR_B->BusInput1 = inst->in;

  /* BusSelector: '<S2>/BusConversion_InsertedFor_Bus Creator_at_inport_0' */
  AC_PFPDR_B->bStartTrigger = AC_PFPDR_B->BusInput1.bStartTrigger;
  for (i = 0; i < 25; i++) {
    AC_PFPDR_B->rT_EG_Act[i] = AC_PFPDR_B->BusInput1.rT_EG_Act[i];
    AC_PFPDR_B->rCA_IP_Act[i] = AC_PFPDR_B->BusInput1.rCA_IP_Act[i];
  }

  rtb_iNum_Cyl = AC_PFPDR_B->BusInput1.iNum_Cyl;
  AC_PFPDR_B->bMisfLim = AC_PFPDR_B->BusInput1.bMisfLim;
  AC_PFPDR_B->bManAbort = AC_PFPDR_B->BusInput1.bManAbort;
  AC_PFPDR_B->bReset = AC_PFPDR_B->BusInput1.bReset;
  AC_PFPDR_B->rLam_Act = AC_PFPDR_B->BusInput1.rLam_Act;
  AC_PFPDR_B->bSteadyState = AC_PFPDR_B->BusInput1.bSteadyState;

  /* End of BusSelector: '<S2>/BusConversion_InsertedFor_Bus Creator_at_inport_0' */

  /* UnitDelay: '<S5>/Unit Delay' */
  AC_PFPDR_B->UnitDelay = AC_PFPDR_DWork->UnitDelay_DSTATE;

  /* UnitDelay: '<S5>/Unit Delay1' */
  AC_PFPDR_B->UnitDelay1 = AC_PFPDR_DWork->UnitDelay1_DSTATE;

  /* S-Function (bur_bus_in): '<S2>/Bus Input' */
  AC_PFPDR_B->BusInput = inst->par;

  /* BusSelector: '<S2>/BusConversion_InsertedFor_Bus Creator_at_inport_1' */
  AC_PFPDR_B->rCA_IP_MaxLim = AC_PFPDR_B->BusInput.rCA_IP_MaxLim;
  AC_PFPDR_B->rT_EG_DevLim = AC_PFPDR_B->BusInput.rT_EG_DevLim;
  AC_PFPDR_B->rCA_IP_EGT = AC_PFPDR_B->BusInput.rCA_IP_EGT;
  rtb_rT_Abort_Delay = AC_PFPDR_B->BusInput.rT_Abort_Delay;

  /* Product: '<S5>/Divide' incorporates:
   *  Constant: '<S5>/Constant'
   */
  AC_PFPDR_B->Divide = AC_PFPDR_B->BusInput.rTi_EGT_Delay / 0.01F;

  /* Product: '<S5>/Product' incorporates:
   *  Constant: '<S5>/Constant'
   */
  AC_PFPDR_B->Product = AC_PFPDR_B->BusInput.rCA_IP_DR_SR * 0.01F;

  /* Product: '<S5>/Product1' incorporates:
   *  Constant: '<S5>/Constant'
   */
  AC_PFPDR_B->Product1 = AC_PFPDR_B->BusInput.rLam_DR_SR * 0.01F;

  /* Product: '<S5>/Product2' incorporates:
   *  Constant: '<S5>/Constant'
   */
  AC_PFPDR_B->Product2 = AC_PFPDR_B->BusInput.rCA_IP_DR_SR_Return * 0.01F;

  /* Product: '<S5>/Product3' incorporates:
   *  Constant: '<S5>/Constant'
   */
  AC_PFPDR_B->Product3 = AC_PFPDR_B->BusInput.rLam_DR_SR_Return * 0.01F;

  /* UnitDelay: '<S5>/Unit Delay2' */
  AC_PFPDR_B->UnitDelay2 = AC_PFPDR_DWork->UnitDelay2_DSTATE;

  /* Saturate: '<S5>/1-24 Cylinder' */
  if (rtb_iNum_Cyl >= 24) {
    AC_PFPDR_B->u4Cylinder = 24U;
  } else if (rtb_iNum_Cyl <= 1) {
    AC_PFPDR_B->u4Cylinder = 1U;
  } else {
    AC_PFPDR_B->u4Cylinder = rtb_iNum_Cyl;
  }

  /* End of Saturate: '<S5>/1-24 Cylinder' */

  /* Chart: '<S5>/Chart (MATLAB)' */
  /* Gateway: SimuBlock/PFPDR_Autocode/PFPDR/Chart (MATLAB) */
  /* During: SimuBlock/PFPDR_Autocode/PFPDR/Chart (MATLAB) */
  if (AC_PFPDR_DWork->is_active_c6_AC_PFPDR == 0U) {
    /* Entry: SimuBlock/PFPDR_Autocode/PFPDR/Chart (MATLAB) */
    AC_PFPDR_DWork->is_active_c6_AC_PFPDR = 1U;

    /* Entry Internal: SimuBlock/PFPDR_Autocode/PFPDR/Chart (MATLAB) */
    /* Transition: '<S7>:2' */
    AC_PFPDR_DWork->is_c6_AC_PFPDR = AC_PFPDR_IN_IDLE;

    /* Entry 'IDLE': '<S7>:1' */
    AC_PFPDR_B->iState = 0;
    AC_PFPDR_B->bLeanox_Man = FALSE;
    AC_PFPDR_B->bPFPDR_active = FALSE;
    AC_PFPDR_B->bEGTSR_active = FALSE;
  } else {
    switch (AC_PFPDR_DWork->is_c6_AC_PFPDR) {
     case AC_PFPDR_IN_Abort:
      /* During 'Abort': '<S7>:65' */
      /* Transition: '<S7>:68' */
      AC_PFPDR_DWork->is_c6_AC_PFPDR = AC_PFPDR_IN_IDLE;

      /* Entry 'IDLE': '<S7>:1' */
      AC_PFPDR_B->iState = 0;
      AC_PFPDR_B->bLeanox_Man = FALSE;
      AC_PFPDR_B->bPFPDR_active = FALSE;
      AC_PFPDR_B->bEGTSR_active = FALSE;
      break;

     case AC_PFPDR_IN_DetectionRun:
      /* During 'DetectionRun': '<S7>:7' */
      if (AC_PFPDR_DWork->bDR_Done) {
        /* Transition: '<S7>:6' */
        /* Exit Internal 'DetectionRun': '<S7>:7' */
        switch (AC_PFPDR_DWork->is_DetectionRun) {
         case AC_PFPDR_IN_IgnpointReturn:
          /* Exit 'IgnpointReturn': '<S7>:71' */
          AC_PFPDR_B->rCA_IP_DR_Offs = 0.0F;
          AC_PFPDR_DWork->bDR_Lam = TRUE;
          AC_PFPDR_DWork->is_DetectionRun = AC_PFPDR_IN_NO_ACTIVE_CHILD;
          break;

         case AC_PFPDR_IN_LambdaReturn:
          /* Exit 'LambdaReturn': '<S7>:70' */
          AC_PFPDR_DWork->bDR_Lam = FALSE;
          AC_PFPDR_B->rLam_DR_Offs = 0.0F;
          AC_PFPDR_DWork->bDR_Done = TRUE;
          AC_PFPDR_B->bLeanox_Man = FALSE;
          AC_PFPDR_DWork->is_DetectionRun = AC_PFPDR_IN_NO_ACTIVE_CHILD;
          break;

         default:
          AC_PFPDR_DWork->is_DetectionRun = AC_PFPDR_IN_NO_ACTIVE_CHILD;
          break;
        }

        AC_PFPDR_DWork->is_c6_AC_PFPDR = AC_PFPDR_IN_EGTSR;

        /* Entry 'EGTSR': '<S7>:5' */
        /*  INIT routine */
        AC_PFPDR_B->iState = 2;
        AC_PFPDR_B->iSubState = 0;
        AC_PFPDR_DWork->iCnt = 0.0F;
        AC_PFPDR_DWork->bEGT_Done = FALSE;
        AC_PFPDR_B->bEGTSR_active = TRUE;
        AC_PFPDR_B->bPFPDR_active = FALSE;

        /*  CYCLIC routine */
      } else if (AC_PFPDR_B->bReset) {
        /* Transition: '<S7>:86' */
        /* Exit Internal 'DetectionRun': '<S7>:7' */
        switch (AC_PFPDR_DWork->is_DetectionRun) {
         case AC_PFPDR_IN_IgnpointReturn:
          /* Exit 'IgnpointReturn': '<S7>:71' */
          AC_PFPDR_B->rCA_IP_DR_Offs = 0.0F;
          AC_PFPDR_DWork->bDR_Lam = TRUE;
          AC_PFPDR_DWork->is_DetectionRun = AC_PFPDR_IN_NO_ACTIVE_CHILD;
          break;

         case AC_PFPDR_IN_LambdaReturn:
          /* Exit 'LambdaReturn': '<S7>:70' */
          AC_PFPDR_DWork->bDR_Lam = FALSE;
          AC_PFPDR_B->rLam_DR_Offs = 0.0F;
          AC_PFPDR_DWork->bDR_Done = TRUE;
          AC_PFPDR_B->bLeanox_Man = FALSE;
          AC_PFPDR_DWork->is_DetectionRun = AC_PFPDR_IN_NO_ACTIVE_CHILD;
          break;

         default:
          AC_PFPDR_DWork->is_DetectionRun = AC_PFPDR_IN_NO_ACTIVE_CHILD;
          break;
        }

        AC_PFPDR_DWork->is_c6_AC_PFPDR = AC_PFPDR_IN_Abort;

        /* Entry 'Abort': '<S7>:65' */
        /*  INIT routine */
        AC_PFPDR_B->iState = 3;
        AC_PFPDR_B->bLeanox_Man = FALSE;
        AC_PFPDR_B->rCA_IP_DR_Offs = 0.0F;
        AC_PFPDR_B->rLam_DR_Offs = 0.0F;
      } else {
        if (AC_PFPDR_B->UnitDelay1) {
          for (i = 0; i < 25; i++) {
            AC_PFPDR_DWork->rCA_IgnP_Act_Filt[i] += AC_PFPDR_B->rCA_IP_Act[i];
          }

          AC_PFPDR_DWork->rCnt_Filt++;
        } else {
          for (i = 0; i < 25; i++) {
            AC_PFPDR_DWork->rCA_IgnP_Act_Filt[i] = AC_PFPDR_B->rCA_IP_Act[i];
          }

          AC_PFPDR_DWork->rCnt_Filt = 1.0F;
        }

        switch (AC_PFPDR_DWork->is_DetectionRun) {
         case AC_PFPDR_IN_Detection:
          /* During 'Detection': '<S7>:10' */
          /* Transition: '<S7>:11' */
          AC_PFPDR_DWork->is_DetectionRun = AC_PFPDR_IN_IgnitionPoint;

          /* Entry 'IgnitionPoint': '<S7>:9' */
          AC_PFPDR_B->iSubState = 2;
          break;

         case AC_PFPDR_IN_IgnitionPoint:
          /* During 'IgnitionPoint': '<S7>:9' */
          if (AC_PFPDR_B->UnitDelay || AC_PFPDR_B->bManAbort) {
            /* Transition: '<S7>:8' */
            AC_PFPDR_DWork->is_DetectionRun = AC_PFPDR_IN_SaveProfile;
            AC_PFP_enter_atomic_SaveProfile(AC_PFPDR_B, AC_PFPDR_DWork, inst);
          } else if (AC_PFPDR_DWork->bDR_Lam || (!AC_PFPDR_B->UnitDelay2)) {
            /* Transition: '<S7>:16' */
            AC_PFPDR_DWork->is_DetectionRun = AC_PFPDR_IN_Lambda;

            /* Entry 'Lambda': '<S7>:15' */
            AC_PFPDR_B->iSubState = 3;
            AC_PFPDR_B->bLeanox_Man = TRUE;
          } else {
            rCA_IP_Max = AC_PFPDR_B->rCA_IP_Act[1];
            i = (int32_T)((uint32_T)AC_PFPDR_B->u4Cylinder + 1U);
            if ((uint32_T)i > 255U) {
              i = 255;
            }

            for (rtb_iNum_Cyl = 2U; rtb_iNum_Cyl <= (uint8_T)i; rtb_iNum_Cyl =
                 (uint8_T)((uint32_T)rtb_iNum_Cyl + 1U)) {
              if (rCA_IP_Max < AC_PFPDR_B->rCA_IP_Act[rtb_iNum_Cyl - 1]) {
                rCA_IP_Max = AC_PFPDR_B->rCA_IP_Act[rtb_iNum_Cyl - 1];
              }
            }

            AC_PFPDR_DWork->bDR_Lam = ((rCA_IP_Max >= AC_PFPDR_B->rCA_IP_MaxLim)
              || AC_PFPDR_B->bMisfLim);
            AC_PFPDR_B->rCA_IP_DR_Offs += AC_PFPDR_B->Product;
          }
          break;

         case AC_PFPDR_IN_IgnpointReturn:
          /* During 'IgnpointReturn': '<S7>:71' */
          if (AC_PFPDR_B->rCA_IP_DR_Offs <= 0.0F) {
            /* Transition: '<S7>:73' */
            /* Exit 'IgnpointReturn': '<S7>:71' */
            AC_PFPDR_B->rCA_IP_DR_Offs = 0.0F;
            AC_PFPDR_DWork->bDR_Lam = TRUE;
            AC_PFPDR_DWork->is_DetectionRun = AC_PFPDR_IN_LambdaReturn;

            /* Entry 'LambdaReturn': '<S7>:70' */
            AC_PFPDR_B->iSubState = 5;
          } else {
            AC_PFPDR_B->rCA_IP_DR_Offs -= AC_PFPDR_B->Product2;
          }
          break;

         case AC_PFPDR_IN_Lambda:
          /* During 'Lambda': '<S7>:15' */
          if (AC_PFPDR_B->UnitDelay || AC_PFPDR_B->bManAbort) {
            /* Transition: '<S7>:17' */
            AC_PFPDR_DWork->is_DetectionRun = AC_PFPDR_IN_SaveProfile;
            AC_PFP_enter_atomic_SaveProfile(AC_PFPDR_B, AC_PFPDR_DWork, inst);
          } else if (AC_PFPDR_B->UnitDelay2 && (!AC_PFPDR_DWork->bDR_Lam)) {
            /* Transition: '<S7>:82' */
            AC_PFPDR_DWork->is_DetectionRun = AC_PFPDR_IN_IgnitionPoint;

            /* Entry 'IgnitionPoint': '<S7>:9' */
            AC_PFPDR_B->iSubState = 2;
          } else {
            AC_PFPDR_B->rLam_DR_Offs -= AC_PFPDR_B->Product1;
          }
          break;

         case AC_PFPDR_IN_LambdaReturn:
          /* During 'LambdaReturn': '<S7>:70' */
          if ((AC_PFPDR_B->rLam_DR_Offs >= 0.0F) || (!AC_PFPDR_DWork->bDR_Lam))
          {
            /* Transition: '<S7>:72' */
            /* Exit 'LambdaReturn': '<S7>:70' */
            AC_PFPDR_DWork->bDR_Lam = FALSE;
            AC_PFPDR_B->rLam_DR_Offs = 0.0F;
            AC_PFPDR_DWork->bDR_Done = TRUE;
            AC_PFPDR_B->bLeanox_Man = FALSE;
            AC_PFPDR_DWork->is_DetectionRun = AC_PFPDR_IN_Detection;

            /* Entry 'Detection': '<S7>:10' */
            AC_PFPDR_B->iSubState = 1;
          } else {
            AC_PFPDR_B->rLam_DR_Offs += AC_PFPDR_B->Product3;
            if (AC_PFPDR_DWork->rLam_bDR < AC_PFPDR_B->rLam_Act) {
              AC_PFPDR_DWork->bDR_Lam = FALSE;
            }
          }
          break;

         default:
          /* During 'SaveProfile': '<S7>:74' */
          /* Transition: '<S7>:75' */
          AC_PFPDR_DWork->is_DetectionRun = AC_PFPDR_IN_IgnpointReturn;

          /* Entry 'IgnpointReturn': '<S7>:71' */
          AC_PFPDR_B->iSubState = 6;
          break;
        }
      }
      break;

     case AC_PFPDR_IN_EGTSR:
      /* During 'EGTSR': '<S7>:5' */
      if (AC_PFPDR_DWork->bEGT_Done) {
        /* Transition: '<S7>:4' */
        AC_PFPDR_exit_atomic_EGTSR(AC_PFPDR_B, inst);
        AC_PFPDR_DWork->is_c6_AC_PFPDR = AC_PFPDR_IN_IDLE;

        /* Entry 'IDLE': '<S7>:1' */
        AC_PFPDR_B->iState = 0;
        AC_PFPDR_B->bLeanox_Man = FALSE;
        AC_PFPDR_B->bPFPDR_active = FALSE;
        AC_PFPDR_B->bEGTSR_active = FALSE;
      } else if (AC_PFPDR_B->bManAbort || AC_PFPDR_B->bReset) {
        /* Transition: '<S7>:67' */
        AC_PFPDR_exit_atomic_EGTSR(AC_PFPDR_B, inst);
        AC_PFPDR_DWork->is_c6_AC_PFPDR = AC_PFPDR_IN_Abort;

        /* Entry 'Abort': '<S7>:65' */
        /*  INIT routine */
        AC_PFPDR_B->iState = 3;
        AC_PFPDR_B->bLeanox_Man = FALSE;
        AC_PFPDR_B->rCA_IP_DR_Offs = 0.0F;
        AC_PFPDR_B->rLam_DR_Offs = 0.0F;
      } else {
        AC_PFPDR_DWork->iCnt++;
        AC_PFPDR_DWork->bEGT_Done = ((AC_PFPDR_DWork->iCnt > AC_PFPDR_B->Divide)
          && AC_PFPDR_B->bSteadyState);

        /*  EXIT routine */
      }
      break;

     default:
      /* During 'IDLE': '<S7>:1' */
      if (AC_PFPDR_B->bStartTrigger && AC_PFPDR_B->bSteadyState) {
        /* Transition: '<S7>:3' */
        AC_PFPDR_DWork->is_c6_AC_PFPDR = AC_PFPDR_IN_DetectionRun;

        /* Entry 'DetectionRun': '<S7>:7' */
        /*  INIT routine */
        AC_PFPDR_B->iState = 1;
        AC_PFPDR_B->bPFPDR_active = TRUE;
        AC_PFPDR_DWork->bDR_Done = FALSE;
        AC_PFPDR_DWork->bDR_Lam = FALSE;
        AC_PFPDR_B->bLeanox_Man = FALSE;
        AC_PFPDR_B->rCA_IP_DR_Offs = 0.0F;
        AC_PFPDR_B->rLam_DR_Offs = 0.0F;
        AC_PFPDR_B->rCA_IP_bDR_Avg = 0.0F;
        i = (int32_T)((uint32_T)AC_PFPDR_B->u4Cylinder + 1U);
        if ((uint32_T)i > 255U) {
          i = 255;
        }

        for (rtb_iNum_Cyl = 2U; rtb_iNum_Cyl <= (uint8_T)i; rtb_iNum_Cyl =
             (uint8_T)((uint32_T)rtb_iNum_Cyl + 1U)) {
          AC_PFPDR_B->rCA_IP_bDR_Avg += AC_PFPDR_B->rCA_IP_Act[rtb_iNum_Cyl - 1];
        }

        AC_PFPDR_B->rCA_IP_bDR_Avg /= (real32_T)AC_PFPDR_B->u4Cylinder;
        AC_PFPDR_DWork->rLam_bDR = AC_PFPDR_B->rLam_Act;
        for (i = 0; i < 25; i++) {
          AC_PFPDR_B->rCA_IP_bDR[i] = AC_PFPDR_B->rCA_IP_Act[i];
          AC_PFPDR_B->rCA_IP_aDR_Offs[i] = 0.0F;
          AC_PFPDR_DWork->rCA_IgnP_Act_Filt[i] = AC_PFPDR_B->rCA_IP_Act[i];
        }

        AC_PFPDR_DWork->rCnt_Filt = 1.0F;

        /* Entry Internal 'DetectionRun': '<S7>:7' */
        /* Transition: '<S7>:58' */
        AC_PFPDR_DWork->is_DetectionRun = AC_PFPDR_IN_Detection;

        /* Entry 'Detection': '<S7>:10' */
        AC_PFPDR_B->iSubState = 1;
      }
      break;
    }
  }

  /* End of Chart: '<S5>/Chart (MATLAB)' */

  /* BusCreator: '<S2>/BusConversion_InsertedFor_Bus Output_at_inport_0' incorporates:
   *  Logic: '<S2>/ZylOpt deact'
   *  SignalConversion: '<S2>/BusConversion_InsertedFor_Bus Output_at_inport_0'
   */
  AC_PFPDR_B->BusConversion_InsertedFor_BusOu.iState[0] = AC_PFPDR_B->iState;
  AC_PFPDR_B->BusConversion_InsertedFor_BusOu.iState[1] = AC_PFPDR_B->iSubState;
  AC_PFPDR_B->BusConversion_InsertedFor_BusOu.rLam_DR_Offs =
    AC_PFPDR_B->rLam_DR_Offs;
  AC_PFPDR_B->BusConversion_InsertedFor_BusOu.rCA_IP_DR_Offs =
    AC_PFPDR_B->rCA_IP_DR_Offs;
  AC_PFPDR_B->BusConversion_InsertedFor_BusOu.bLeanox_Man =
    AC_PFPDR_B->bLeanox_Man;
  for (i = 0; i < 25; i++) {
    AC_PFPDR_B->BusConversion_InsertedFor_BusOu.rCA_IP_DR_Profile[i] =
      AC_PFPDR_B->rCA_IP_aDR_Offs[i];
    AC_PFPDR_B->BusConversion_InsertedFor_BusOu.rCA_IP_EGT_Profile[i] =
      AC_PFPDR_B->rCA_IP_EGT_Offs[i];
  }

  AC_PFPDR_B->BusConversion_InsertedFor_BusOu.bPFPDR_act =
    AC_PFPDR_B->bPFPDR_active;
  AC_PFPDR_B->BusConversion_InsertedFor_BusOu.bEGTSR_act =
    AC_PFPDR_B->bEGTSR_active;
  AC_PFPDR_B->BusConversion_InsertedFor_BusOu.bZYLOPT_OFF =
    (AC_PFPDR_B->bPFPDR_active || AC_PFPDR_B->bEGTSR_active);

  /* End of BusCreator: '<S2>/BusConversion_InsertedFor_Bus Output_at_inport_0' */

  /* S-Function (bur_bus_out): '<S2>/Bus Output' */
  inst->out = AC_PFPDR_B->BusConversion_InsertedFor_BusOu;

  /* MATLAB Function: '<S6>/Abort Condition 1' */
  /* MATLAB Function 'SimuBlock/PFPDR_Autocode/PFPDR/Abort Conditions/Abort Condition 1': '<S10>:1' */
  /* variable array size not suported by autocode: */
  /* abort1 = (sum((rCA_Knck_Red(1:iNum_Cyl)-min(rCA_Knck_Red(1:iNum_Cyl)))>0)/iNum_Cyl) >= 0.25; */
  /*  rCA_Knck_Red_min = rCA_Knck_Red(2); */
  /*  for iCyl=2:iNum_Cyl+1 */
  /*       if rCA_Knck_Red_min > rCA_Knck_Red(iCyl) */
  /*           rCA_Knck_Red_min = rCA_Knck_Red(iCyl); */
  /*       end */
  /*  end */
  /* '<S10>:1:10' */
  rCA_IP_Max = 0.0F;

  /* '<S10>:1:11' */
  i = (int32_T)((uint32_T)AC_PFPDR_B->u4Cylinder + 1U);
  if ((uint32_T)i > 255U) {
    i = 255;
  }

  /* '<S10>:1:11' */
  for (rtb_iNum_Cyl = 2U; rtb_iNum_Cyl <= (uint8_T)i; rtb_iNum_Cyl = (uint8_T)
       ((uint32_T)rtb_iNum_Cyl + 1U)) {
    /* '<S10>:1:11' */
    if (AC_PFPDR_B->BusInput1.rCA_Knck_Red[rtb_iNum_Cyl - 1] > 0.0F) {
      /* '<S10>:1:12' */
      /* '<S10>:1:13' */
      rCA_IP_Max++;
    }
  }

  if (rCA_IP_Max >= (real32_T)(uint8_T)(int32_T)rt_roundd(0.25 * (real_T)
       AC_PFPDR_B->u4Cylinder, inst)) {
    /* '<S10>:1:16' */
    /* '<S10>:1:17' */
    rtb_abort1 = TRUE;
  } else {
    /* '<S10>:1:19' */
    rtb_abort1 = FALSE;
  }

  /* End of MATLAB Function: '<S6>/Abort Condition 1' */

  /* Switch: '<S6>/Switch' incorporates:
   *  Constant: '<S6>/AlterMotor'
   *  Constant: '<S6>/NeuerMotor '
   */
  if (AC_PFPDR_B->BusInput1.bPFPDR_Profile) {
    rtb_Switch = 5;
  } else {
    rtb_Switch = 4;
  }

  /* End of Switch: '<S6>/Switch' */

  /* MATLAB Function: '<S6>/Abort Condition 2' */
  /* MATLAB Function 'SimuBlock/PFPDR_Autocode/PFPDR/Abort Conditions/Abort Condition 2': '<S11>:1' */
  /* variable array size not suported by autocode: */
  /* abort2 = sum((rCA_IgnP_Set - rCA_Ign_Act(1:iNum_Cyl)) >= rCA_Dev_Max)>0; */
  /* '<S11>:1:4' */
  rtb_abort2 = FALSE;

  /* '<S11>:1:5' */
  i = (int32_T)((uint32_T)AC_PFPDR_B->u4Cylinder + 1U);
  if ((uint32_T)i > 255U) {
    i = 255;
  }

  /* '<S11>:1:5' */
  for (rtb_iNum_Cyl = 2U; rtb_iNum_Cyl <= (uint8_T)i; rtb_iNum_Cyl = (uint8_T)
       ((uint32_T)rtb_iNum_Cyl + 1U)) {
    /* '<S11>:1:5' */
    if ((real_T)(AC_PFPDR_B->BusInput1.rCA_IP_Set - AC_PFPDR_B->
                 rCA_IP_Act[rtb_iNum_Cyl - 1]) >= (real_T)rtb_Switch) {
      /* '<S11>:1:6' */
      /* '<S11>:1:7' */
      rtb_abort2 = TRUE;
    }
  }

  /* End of MATLAB Function: '<S6>/Abort Condition 2' */

  /* MATLAB Function: '<S6>/Abort Condition 3' */
  /* MATLAB Function 'SimuBlock/PFPDR_Autocode/PFPDR/Abort Conditions/Abort Condition 3': '<S12>:1' */
  /* '<S12>:1:4' */
  rtb_abort3 = (AC_PFPDR_B->rLam_DR_Offs <= -AC_PFPDR_B->BusInput.rLam_DR_Lim);

  /* BusCreator: '<S2>/BusConversion_InsertedFor_Bus Output1_at_inport_0' incorporates:
   *  SignalConversion: '<S2>/BusConversion_InsertedFor_Bus Output1_at_inport_0'
   */
  AC_PFPDR_B->BusConversion_InsertedFor_Bus_c.rT_Sampling = 0.01F;
  for (i = 0; i < 25; i++) {
    AC_PFPDR_B->BusConversion_InsertedFor_Bus_c.rCA_IP_aDR[i] =
      AC_PFPDR_B->rCA_IP_aDR[i];
    AC_PFPDR_B->BusConversion_InsertedFor_Bus_c.rCA_IP_bDR[i] =
      AC_PFPDR_B->rCA_IP_bDR[i];
  }

  AC_PFPDR_B->BusConversion_InsertedFor_Bus_c.rCA_IP_aDR_Avg =
    AC_PFPDR_B->rCA_IP_aDR_Max;
  AC_PFPDR_B->BusConversion_InsertedFor_Bus_c.rCA_IP_bDR_Avg =
    AC_PFPDR_B->rCA_IP_bDR_Avg;
  AC_PFPDR_B->BusConversion_InsertedFor_Bus_c.bAbort_DR[0] = rtb_abort1;
  AC_PFPDR_B->BusConversion_InsertedFor_Bus_c.bAbort_DR[1] = rtb_abort2;
  AC_PFPDR_B->BusConversion_InsertedFor_Bus_c.bAbort_DR[2] = rtb_abort3;

  /* End of BusCreator: '<S2>/BusConversion_InsertedFor_Bus Output1_at_inport_0' */

  /* S-Function (bur_bus_out): '<S2>/Bus Output1' */
  inst->dbg = AC_PFPDR_B->BusConversion_InsertedFor_Bus_c;

  /* Logic: '<S6>/Abort' */
  rtb_Abort = (rtb_abort1 || rtb_abort2 || rtb_abort3);

  /* Switch: '<S8>/Switch3' incorporates:
   *  Abs: '<S5>/Abs'
   *  Constant: '<S5>/TRUE'
   *  Logic: '<S5>/Logical Operator'
   *  RelationalOperator: '<S8>/groesser '
   *  RelationalOperator: '<S8>/kleiner'
   *  Sum: '<S5>/plus '
   *  Switch: '<S8>/Switch1'
   *  Switch: '<S8>/Switch2'
   *  UnitDelay: '<S8>/Unit Delay2'
   */
  if (!AC_PFPDR_B->bPFPDR_active) {
    rtb_abort1 = TRUE;
  } else if (AC_PFPDR_B->BusInput1.rPos_CBV < AC_PFPDR_B->BusInput.rPos_CBV_Opt)
  {
    /* Switch: '<S8>/Switch1' incorporates:
     *  Constant: '<S8>/FALSE'
     */
    rtb_abort1 = FALSE;
  } else if (AC_PFPDR_B->BusInput1.rPos_CBV > AC_PFPDR_B->BusInput.rPos_CBV_Opt
             + (real32_T)fabs(AC_PFPDR_B->BusInput.rPos_CBV_Hys)) {
    /* Switch: '<S8>/Switch2' incorporates:
     *  Constant: '<S8>/TRUE'
     *  Switch: '<S8>/Switch1'
     */
    rtb_abort1 = TRUE;
  } else {
    rtb_abort1 = AC_PFPDR_DWork->UnitDelay2_DSTATE_l;
  }

  /* End of Switch: '<S8>/Switch3' */

  /* Sum: '<S9>/Subtract' */
  rtb_Subtract = rtb_rT_Abort_Delay - AC_PFPDR_B->BusInput.rT_Abort_Filter;

  /* Outputs for Atomic SubSystem: '<S9>/TON' */
  AC_PFPDR_TON(rtb_Abort, rtb_rT_Abort_Delay, &AC_PFPDR_B->TON,
               &AC_PFPDR_DWork->TON, inst);

  /* End of Outputs for SubSystem: '<S9>/TON' */

  /* Outputs for Atomic SubSystem: '<S9>/TON1' */
  AC_PFPDR_TON(rtb_Abort, rtb_Subtract, &AC_PFPDR_B->TON1, &AC_PFPDR_DWork->TON1, inst);

  /* End of Outputs for SubSystem: '<S9>/TON1' */

  /* Update for UnitDelay: '<S5>/Unit Delay' */
  AC_PFPDR_DWork->UnitDelay_DSTATE = AC_PFPDR_B->TON.LogicalOperator3;

  /* Update for UnitDelay: '<S5>/Unit Delay1' */
  AC_PFPDR_DWork->UnitDelay1_DSTATE = AC_PFPDR_B->TON1.LogicalOperator3;

  /* Update for UnitDelay: '<S5>/Unit Delay2' */
  AC_PFPDR_DWork->UnitDelay2_DSTATE = rtb_abort1;

  /* Update for UnitDelay: '<S8>/Unit Delay2' */
  AC_PFPDR_DWork->UnitDelay2_DSTATE_l = rtb_abort1;
}

/* Model initialize function */
void AC_PFPDR_initialize(struct PFPDR* inst)
{
  /* (no initialization code required) */
}

/* Model terminate function */
void AC_PFPDR_terminate(struct PFPDR* inst)
{
  /* (no terminate code required) */
}

/*======================== TOOL VERSION INFORMATION ==========================*
 * MATLAB 8.0 (R2012b)20-Jul-2012                                             *
 * Simulink 8.0 (R2012b)20-Jul-2012                                           *
 * Simulink Coder 8.3 (R2012b)20-Jul-2012                                     *
 * Embedded Coder 6.3 (R2012b)20-Jul-2012                                     *
 * Stateflow 8.0 (R2012b)20-Jul-2012                                          *
 *============================================================================*/

/*======================= LICENSE IN USE INFORMATION =========================*
 * matlab                                                                     *
 * matlab_coder                                                               *
 * real-time_workshop                                                         *
 * rtw_embedded_coder                                                         *
 * simulink                                                                   *
 * stateflow                                                                  *
 *============================================================================*/
```

#### main.c
```c
/********************************************************************
 * COPYRIGHT -- Bernecker + Rainer Industrie-Elektronik Ges.m.b.H.
 ********************************************************************
 * Program: AC_PFPDR
 * File: main.c
 * Author: 502423184
 * Created: Fri Apr 24 12:55:11 2015
 ********************************************************************
 * Implementation of program AC_PFPDR
 ********************************************************************
 * Generated with B&R Automation Studio Target for Simulink V4.2
 * (ERT based)
 ********************************************************************/
#include <bur/plctypes.h>
#include "AC_PFPDR.h"
#include "rtwtypes.h"

/* Defines */
#define SS_TERMINATE 4
#define SS_OUTPUT 3
#define SS_INITIALIZE 2

/*  Data Types */

/**************************** GLOBAL DATA *************************************/
/*  Definitions */

/*  Declarations  */

/***************************** FILE SCOPE DATA ********************************/

/*************************** FUNCTIONS ****************************************/
#ifdef __cplusplus

unsigned long bur_heap_size = 6553500;

#endif

void PFPDR(struct PFPDR* inst)
{
  BlockIO_AC_PFPDR *AC_PFPDR_B = &(inst)->bur_BlockIO_AC_PFPDR;
	D_Work_AC_PFPDR *AC_PFPDR_DWork = &(inst)->bur_D_Work_AC_PFPDR;

  switch (inst->ssMethodType)
  {
   case SS_INITIALIZE:
    /* call model initialize function */
    AC_PFPDR_initialize(inst);
    break;

   case SS_OUTPUT:
    /* call model step function */
    AC_PFPDR_step(AC_PFPDR_B, AC_PFPDR_DWork, inst);

    break;

   case SS_TERMINATE:
    /* call model terminate function */
    AC_PFPDR_terminate(inst);
    break;
  }
}

/*****************************************************************************
   Function block sample time: 0.01s
 *****************************************************************************/

/*****************************************************************************
   B&R Automation Studio Target for Simulink Version: A4.4.1 (09-Dec-2014)
 *****************************************************************************/

/*======================== TOOL VERSION INFORMATION ==========================*
 * MATLAB 8.0 (R2012b)20-Jul-2012                                             *
 * Simulink 8.0 (R2012b)20-Jul-2012                                           *
 * Simulink Coder 8.3 (R2012b)20-Jul-2012                                     *
 * Embedded Coder 6.3 (R2012b)20-Jul-2012                                     *
 * Stateflow 8.0 (R2012b)20-Jul-2012                                          *
 *============================================================================*/

/*======================= LICENSE IN USE INFORMATION =========================*
 * matlab                                                                     *
 * matlab_coder                                                               *
 * real-time_workshop                                                         *
 * rtw_embedded_coder                                                         *
 * simulink                                                                   *
 * stateflow                                                                  *
 *============================================================================*/
```

#### lib_properties.txt
```
For manual assignment to hardware configuration please
add the following additional include directories:

\Logical\MATLAB_includes\R2012b\

And the following additional build options:

-lm -D MODEL=AC_PFPDR -D NUMST=1 -D NCSTATES=0 -D HAVESTDIO -D ONESTEPFCN=1 -D TERMFCN=1 -D MAT_FILE=0 -D MULTI_INSTANCE_CODE=1 -D INTEGER_CODE=0 -D MT=0 -D CLASSIC_INTERFACE=0 -D TID01EQ=0
```

### Library Logical/EngineController/Lib_EC/lIP_EGTCtr (ANSIC)

#### lIP_EGTCtr.fun
```iecst
FUNCTION_BLOCK fIP_EGTCtr
  VAR_INPUT
    ssMethodType: SINT;
  END_VAR  VAR_INPUT
        in : tEGTCtr_In; (**)
  END_VAR
  VAR_INPUT
        perm : tEGTCtr_Perm; (**)
  END_VAR
 VAR_OUTPUT
        out : tEGTCtr_Out; (**)
  END_VAR
	VAR
		bur_BlockIO_IP_EGTCtr : BlockIO_IP_EGTCtr;
	END_VAR
	VAR
		bur_D_Work_IP_EGTCtr : D_Work_IP_EGTCtr;
	END_VAR
END_FUNCTION_BLOCK
```
